// TIA Portal project "Robot_Presantation_Project_V1.0" (V16)

(* hardware
DEVICE "S7-1200 station_1"  S7-1200 Station
   slot 0: "Rack_0"  S7-1200 Rack  Rack  V1.0
   slot 1: "PLC_1"  CPU 1214C DC/DC/DC  6ES7 214-1AG40-0XB0  V4.4
   slot 2: "DI 16/DQ 16x24VDC_1"  6ES7 223-1BL32-0XB0  V2.0
DEVICE "GSD device_1"  GSD.Device.PN
   slot 0: "Rack"  Rack  V1.0
   slot 0: "RC700-PROFINET-IO"  RT RC700_PNIO_V2  RC700-PROFINET-IO  V1.0
      slot 0: "RT RC700_PNIO_V2"  RT RC700_PNIO_V2
      slot 1: "Interface"  Interface
         slot 1: "RJ45 100 MBit/s"  RJ45 100 MBit/s
   slot 1: "Output 32 bytes_1"  Output 32 bytes
      slot 0: "Output 32 bytes"  Output 32 bytes
   slot 2: "Input 32 bytes_1"  Input 32 bytes
      slot 0: "Input 32 bytes"  Input 32 bytes
*)

// ===== PLC "PLC_1"  CPU 1214C DC/DC/DC =====

VAR_GLOBAL   // PLC tag table "Default tag table"
   "Processing Request" AT %M0.0 : Bool;
   "Button_Led_1" AT %Q0.0 : Bool;
   "Permission_To_Send_Response" AT %M0.1 : Bool;
   "Video_Done_Playing" AT %M50.0 : Bool;
   "Tag_3" AT %M1.0 : Bool;
   "Tag_4" AT %M100.0 : Bool;
   "ROBOT_1_READY" AT %M200.0 : Bool;
   "PLC_Enable_Procedures" AT %M2.0 : Bool;
   "Permission_To_Write_To_PC" AT %M3.0 : Bool;
   "Error_On_Communication" AT %M5.0 : Bool;
   "Reset_Error_On_Communication" AT %M5.1 : Bool;
   "Button_1" AT %I0.0 : Bool;
   "Tag_1" AT %M50.1 : Bool;
   "Button_2" AT %I0.1 : Bool;
   "Button_Led_2" AT %Q0.1 : Bool;
   "Button_3" AT %I0.2 : Bool;
   "Button_Led_3" AT %Q0.2 : Bool;
   "TEST_BIT_ROBOT_1_AT_POSITION" AT %M500.0 : Bool;
   "TEST_BIT_ROBOT_1_AT_HOME" AT %M500.1 : Bool;
   "Virtual Button 1" AT %M600.0 : Bool;
   "Tag_7" AT %M6000.0 : Bool;
   "Toggle_test_Bit_Robot_1_At_position" AT %M500.2 : Bool;
   "ROBOT_AT_POSITION_ID_TEMP" AT %MW33 : Int;
   "Robot_2_Ready" AT %M200.1 : Bool;
   "Enable_Robots" AT %M700.0 : Bool;
   "ROBOT_2_AT_POSITION_ID_TEMP" AT %MW35 : Int;
   "System_Byte" AT %MB299 : Byte;
   "FirstScan" AT %M299.0 : Bool;
   "DiagStatusUpdate" AT %M299.1 : Bool;
   "AlwaysTRUE" AT %M299.2 : Bool;
   "AlwaysFALSE" AT %M299.3 : Bool;
   "Clock_Byte" AT %MB298 : Byte;
   "Clock_10Hz" AT %M298.0 : Bool;
   "Clock_5Hz" AT %M298.1 : Bool;
   "Clock_2.5Hz" AT %M298.2 : Bool;
   "Clock_2Hz" AT %M298.3 : Bool;
   "Clock_1.25Hz" AT %M298.4 : Bool;
   "Clock_1Hz" AT %M298.5 : Bool;
   "Clock_0.625Hz" AT %M298.6 : Bool;
   "Clock_0.5Hz" AT %M298.7 : Bool;
   "Button_4" AT %I0.3 : Bool;
   "Button_5" AT %I0.4 : Bool;
   "Button_6" AT %I0.5 : Bool;
   "Button_7" AT %I0.6 : Bool;
   "Button_8" AT %I0.7 : Bool;
   "Button_9" AT %I1.0 : Bool;
   "Button_10" AT %I1.1 : Bool;
   "Button_11" AT %I1.2 : Bool;
   "Button_12" AT %I1.3 : Bool;
   "Button_13" AT %I1.4 : Bool;
   "Button_14" AT %I1.5 : Bool;
   "Button_15" AT %I1.6 : Bool;
   "Button_16" AT %I1.7 : Bool;
   "Button_17" AT %I2.0 : Bool;
   "Button_18" AT %I2.1 : Bool;
   "Button_Led_4" AT %Q0.3 : Bool;
   "Button_Led_5" AT %Q0.4 : Bool;
   "Button_Led_6" AT %Q0.5 : Bool;
   "Button_Led_7" AT %Q0.6 : Bool;
   "Button_Led_8" AT %Q0.7 : Bool;
   "Button_Led_9" AT %Q1.0 : Bool;
   "Button_Led_10" AT %Q1.1 : Bool;
   "Button_Led_11" AT %Q1.2 : Bool;
   "Button_Led_12" AT %Q1.3 : Bool;
   "Button_Led_13" AT %Q1.4 : Bool;
   "Button_Led_14" AT %Q1.5 : Bool;
   "Button_Led_15" AT %Q1.6 : Bool;
   "Button_Led_16" AT %Q1.7 : Bool;
   "Button_Led_17" AT %Q2.0 : Bool;
   "Button_Led_18" AT %Q2.1 : Bool;
   "Robot_Doors_Latched" AT %M700.1 : Bool;
   "Robot_Latch_Doors" AT %Q3.7 : Bool;
   "Input_Data1_From_Robot" AT %IW68 : Word;
   "Input_Data2_From_Robot" AT %IW70 : Word;
   "Input_Data3_From_Robot" AT %IW72 : Word;
   "Input_Data4_From_Robot" AT %IW74 : Word;
   "Output_Data1_To_Robot" AT %QW64 : Word;
   "Output_Data2_To_Robot" AT %QW66 : Word;
   "Output_Data3_To_Robot" AT %QW68 : Word;
   "EMG_OK" AT %I3.7 : Bool;
   "Robot_Reset_Done" AT %M700.2 : Bool;
   "Robot_HOME_OK" AT %M700.3 : Bool;
   "Tag_2" AT %M1003.0 : Bool;
   "Tag_5" AT %M8000.0 : Bool;
   "Virtual Button 2" AT %M600.1 : Bool;
   "Virtual Button 3" AT %M600.2 : Bool;
   "Virtual Button  4" AT %M600.3 : Bool;
   "Virtual Button 5" AT %M600.4 : Bool;
   "Virtual Button 6" AT %M600.5 : Bool;
   "Virtual Button 7" AT %M6000.6 : Bool;
   "Virtual Button 8" AT %M600.7 : Bool;
   "Virtual Button 9" AT %M601.0 : Bool;
   "Virtual Button 10" AT %M601.1 : Bool;
   "Virtual Button 11" AT %M601.2 : Bool;
   "Virtual Button 12" AT %M601.3 : Bool;
   "Virtual Button 13" AT %M601.4 : Bool;
   "Virtual Button 14" AT %M601.5 : Bool;
   "Virtual Button 15" AT %M601.6 : Bool;
   "Virtual Button 16" AT %M601.7 : Bool;
   "Virtual Button 17" AT %M602.0 : Bool;
   "Virtual Button 18" AT %M602.1 : Bool;
   "Enable All Virtual Buttons" AT %M602.2 : Bool;
END_VAR

DATA_BLOCK "PLC_PC_Handshake"   // DB1
{ S7_Optimized_Access := 'FALSE' }
VERSION : 0.1
   VAR
      PC_To_PLC_Request_Connection : Bool;
      PLC_To_PC_Response_Connection : Bool;
      PC_Ready : Bool;
      PC_Busy : Bool;
      PLC_To_PC_Ready_To_Play_Video_Robot_1 : Bool;
      TestConnection : Bool;
      Connection_To_PC_Lost : Bool;
      PC_To_PLC_Video_Playing_Robot_1 : Bool;
      PC_To_PLC_Video_Done_Playing_Robot_1 : Bool;
      PC_To_PLC_Video_Playing_Robot_2 : Bool;
      PC_To_PLC_Video_Done_Playing_Robot_2 : Bool;
      Buffer_Array_Robot_1 : Array[0..19] of Int;
      Buffer_Array_Robot_2 : Array[0..19] of Int;
      PLC_To_PC_Ready_To_Play_Video_Robot_2 : Bool;
      Empty_Array : Array[0..19] of Int;
   END_VAR
BEGIN
END_DATA_BLOCK

DATA_BLOCK "DB_Robot"   // DB45
{ S7_Optimized_Access := 'FALSE' }
VERSION : 0.1
   VAR
      Ready : Bool;
      Running : Bool;
      Paused : Bool;
      Error : Bool;
      Warning : Bool;
      Inside_Box1 : Bool;
      Inside_Box2 : Bool;
      Inside_Box3 : Bool;
      s1 : Bool;
      s2 : Bool;
      s3 : Bool;
      s4 : Bool;
      s5 : Bool;
      s6 : Bool;
      s7 : Bool;
      s8 : Bool;
      At_Position_ID_Robot_1 : Word;
      ErrorID : Word;
      At_Position_ID_Robot_2 : Word;
      Start : Bool;
      Pause : Bool;
      Continue : Bool;
      Reset : Bool;
      Spare_Out1 : Bool;
      Spare_Out2 : Bool;
      Spare_Out3 : Bool;
      Spare_Out4 : Bool;
      Spare_Out5 : Bool;
      Spare_Out6 : Bool;
      Spare_Out7 : Bool;
      Spare_Out8 : Bool;
      Spare_Out9 : Bool;
      Spare_Out10 : Bool;
      Spare_Out11 : Bool;
      Spare_Out12 : Bool;
      To_Position_ID_Robot_1 : Word;
      To_Position_ID_Robot_2 : Word;
   END_VAR
BEGIN
END_DATA_BLOCK

// folder: DBs From FB

DATA_BLOCK "Button_Number_1"   // DB5
{ S7_Optimized_Access := 'TRUE' }
VERSION : 0.1
// stored: InstanceOfName onButton_Press
"onButton_Press"
BEGIN
END_DATA_BLOCK

DATA_BLOCK "Button_Number_2"   // DB8
{ S7_Optimized_Access := 'TRUE' }
VERSION : 0.1
// stored: InstanceOfName onButton_Press
"onButton_Press"
BEGIN
END_DATA_BLOCK

DATA_BLOCK "Button_Number_3"   // DB10
{ S7_Optimized_Access := 'TRUE' }
VERSION : 0.1
// stored: InstanceOfName onButton_Press
"onButton_Press"
BEGIN
END_DATA_BLOCK

DATA_BLOCK "Robot_1_Control"   // DB11
{ S7_Optimized_Access := 'TRUE' }
VERSION : 0.1
// stored: InstanceOfName Robot_Control
"Robot_Control"
BEGIN
END_DATA_BLOCK

DATA_BLOCK "Robot_2_Control"   // DB12
{ S7_Optimized_Access := 'TRUE' }
VERSION : 0.1
// stored: InstanceOfName Robot_Control
"Robot_Control"
BEGIN
END_DATA_BLOCK

DATA_BLOCK "Button_Number_4"   // DB20
{ S7_Optimized_Access := 'TRUE' }
VERSION : 0.1
// stored: InstanceOfName onButton_Press
"onButton_Press"
BEGIN
END_DATA_BLOCK

DATA_BLOCK "Button_Number_5"   // DB21
{ S7_Optimized_Access := 'TRUE' }
VERSION : 0.1
// stored: InstanceOfName onButton_Press
"onButton_Press"
BEGIN
END_DATA_BLOCK

DATA_BLOCK "Button_Number_6"   // DB22
{ S7_Optimized_Access := 'TRUE' }
VERSION : 0.1
// stored: InstanceOfName onButton_Press
"onButton_Press"
BEGIN
END_DATA_BLOCK

DATA_BLOCK "Button_Number_7"   // DB23
{ S7_Optimized_Access := 'TRUE' }
VERSION : 0.1
// stored: InstanceOfName onButton_Press
"onButton_Press"
BEGIN
END_DATA_BLOCK

DATA_BLOCK "Button_Number_8"   // DB24
{ S7_Optimized_Access := 'TRUE' }
VERSION : 0.1
// stored: InstanceOfName onButton_Press
"onButton_Press"
BEGIN
END_DATA_BLOCK

DATA_BLOCK "Button_Number_9"   // DB25
{ S7_Optimized_Access := 'TRUE' }
VERSION : 0.1
// stored: InstanceOfName onButton_Press
"onButton_Press"
BEGIN
END_DATA_BLOCK

DATA_BLOCK "Button_Number_10"   // DB26
{ S7_Optimized_Access := 'TRUE' }
VERSION : 0.1
// stored: InstanceOfName onButton_Press
"onButton_Press"
BEGIN
END_DATA_BLOCK

DATA_BLOCK "Button_Number_11"   // DB28
{ S7_Optimized_Access := 'TRUE' }
VERSION : 0.1
// stored: InstanceOfName onButton_Press
"onButton_Press"
BEGIN
END_DATA_BLOCK

DATA_BLOCK "Button_Number_12"   // DB30
{ S7_Optimized_Access := 'TRUE' }
VERSION : 0.1
// stored: InstanceOfName onButton_Press
"onButton_Press"
BEGIN
END_DATA_BLOCK

DATA_BLOCK "Button_Number_13"   // DB32
{ S7_Optimized_Access := 'TRUE' }
VERSION : 0.1
// stored: InstanceOfName onButton_Press
"onButton_Press"
BEGIN
END_DATA_BLOCK

DATA_BLOCK "Button_Number_14"   // DB34
{ S7_Optimized_Access := 'TRUE' }
VERSION : 0.1
// stored: InstanceOfName onButton_Press
"onButton_Press"
BEGIN
END_DATA_BLOCK

DATA_BLOCK "Button_Number_15"   // DB36
{ S7_Optimized_Access := 'TRUE' }
VERSION : 0.1
// stored: InstanceOfName onButton_Press
"onButton_Press"
BEGIN
END_DATA_BLOCK

DATA_BLOCK "Button_Number_16"   // DB38
{ S7_Optimized_Access := 'TRUE' }
VERSION : 0.1
// stored: InstanceOfName onButton_Press
"onButton_Press"
BEGIN
END_DATA_BLOCK

DATA_BLOCK "Button_Number_17"   // DB40
{ S7_Optimized_Access := 'TRUE' }
VERSION : 0.1
// stored: InstanceOfName onButton_Press
"onButton_Press"
BEGIN
END_DATA_BLOCK

DATA_BLOCK "Button_Number_18"   // DB42
{ S7_Optimized_Access := 'TRUE' }
VERSION : 0.1
// stored: InstanceOfName onButton_Press
"onButton_Press"
BEGIN
END_DATA_BLOCK

// folder: System blocks/Program resources

DATA_BLOCK "TON_TestConnection_On_Signal"   // DB3
{ S7_Optimized_Access := 'TRUE' }
AUTHOR : Simatic
FAMILY : IEC
NAME : IEC_TMR
VERSION : 1.0
// stored: InstanceOfName IEC_TIMER
"IEC_TIMER"
BEGIN
END_DATA_BLOCK

DATA_BLOCK "TON_TestConnection_Off_Signal"   // DB4
{ S7_Optimized_Access := 'TRUE' }
AUTHOR : Simatic
FAMILY : IEC
NAME : IEC_TMR
VERSION : 1.0
// stored: InstanceOfName IEC_TIMER
"IEC_TIMER"
BEGIN
END_DATA_BLOCK

DATA_BLOCK "Test_Timer_Sequence_1"   // DB6
{ S7_Optimized_Access := 'TRUE' }
AUTHOR : Simatic
FAMILY : IEC
NAME : IEC_TMR
VERSION : 1.0
// stored: InstanceOfName IEC_TIMER
"IEC_TIMER"
BEGIN
END_DATA_BLOCK

DATA_BLOCK "Test_Timer_Sequence_2"   // DB7
{ S7_Optimized_Access := 'TRUE' }
AUTHOR : Simatic
FAMILY : IEC
NAME : IEC_TMR
VERSION : 1.0
// stored: InstanceOfName IEC_TIMER
"IEC_TIMER"
BEGIN
END_DATA_BLOCK

DATA_BLOCK "Test_Timer_Sequence_3"   // DB9
{ S7_Optimized_Access := 'TRUE' }
AUTHOR : Simatic
FAMILY : IEC
NAME : IEC_TMR
VERSION : 1.0
// stored: InstanceOfName IEC_TIMER
"IEC_TIMER"
BEGIN
END_DATA_BLOCK

DATA_BLOCK "Enable_PLC_PC_Comms"   // DB13
{ S7_Optimized_Access := 'TRUE' }
AUTHOR : Simatic
FAMILY : IEC
NAME : IEC_TMR
VERSION : 1.0
// stored: InstanceOfName IEC_TIMER
"IEC_TIMER"
BEGIN
END_DATA_BLOCK

DATA_BLOCK "Test_Timer_Sequence_4"   // DB14
{ S7_Optimized_Access := 'TRUE' }
AUTHOR : Simatic
FAMILY : IEC
NAME : IEC_TMR
VERSION : 1.0
// stored: InstanceOfName IEC_TIMER
"IEC_TIMER"
BEGIN
END_DATA_BLOCK

DATA_BLOCK "Test_Timer_Sequence_5"   // DB15
{ S7_Optimized_Access := 'TRUE' }
AUTHOR : Simatic
FAMILY : IEC
NAME : IEC_TMR
VERSION : 1.0
// stored: InstanceOfName IEC_TIMER
"IEC_TIMER"
BEGIN
END_DATA_BLOCK

DATA_BLOCK "Test_Timer_Sequence_6"   // DB16
{ S7_Optimized_Access := 'TRUE' }
AUTHOR : Simatic
FAMILY : IEC
NAME : IEC_TMR
VERSION : 1.0
// stored: InstanceOfName IEC_TIMER
"IEC_TIMER"
BEGIN
END_DATA_BLOCK

DATA_BLOCK "Test_Timer_Sequence_7"   // DB17
{ S7_Optimized_Access := 'TRUE' }
AUTHOR : Simatic
FAMILY : IEC
NAME : IEC_TMR
VERSION : 1.0
// stored: InstanceOfName IEC_TIMER
"IEC_TIMER"
BEGIN
END_DATA_BLOCK

DATA_BLOCK "Test_Timer_Sequence_8"   // DB18
{ S7_Optimized_Access := 'TRUE' }
AUTHOR : Simatic
FAMILY : IEC
NAME : IEC_TMR
VERSION : 1.0
// stored: InstanceOfName IEC_TIMER
"IEC_TIMER"
BEGIN
END_DATA_BLOCK

DATA_BLOCK "Test_Timer_Sequence_9"   // DB19
{ S7_Optimized_Access := 'TRUE' }
AUTHOR : Simatic
FAMILY : IEC
NAME : IEC_TMR
VERSION : 1.0
// stored: InstanceOfName IEC_TIMER
"IEC_TIMER"
BEGIN
END_DATA_BLOCK

DATA_BLOCK "Test_Timer_Sequence_10"   // DB27
{ S7_Optimized_Access := 'TRUE' }
AUTHOR : Simatic
FAMILY : IEC
NAME : IEC_TMR
VERSION : 1.0
// stored: InstanceOfName IEC_TIMER
"IEC_TIMER"
BEGIN
END_DATA_BLOCK

DATA_BLOCK "Test_Timer_Sequence_11"   // DB29
{ S7_Optimized_Access := 'TRUE' }
AUTHOR : Simatic
FAMILY : IEC
NAME : IEC_TMR
VERSION : 1.0
// stored: InstanceOfName IEC_TIMER
"IEC_TIMER"
BEGIN
END_DATA_BLOCK

DATA_BLOCK "Test_Timer_Sequence_12"   // DB31
{ S7_Optimized_Access := 'TRUE' }
AUTHOR : Simatic
FAMILY : IEC
NAME : IEC_TMR
VERSION : 1.0
// stored: InstanceOfName IEC_TIMER
"IEC_TIMER"
BEGIN
END_DATA_BLOCK

DATA_BLOCK "Test_Timer_Sequence_13"   // DB33
{ S7_Optimized_Access := 'TRUE' }
AUTHOR : Simatic
FAMILY : IEC
NAME : IEC_TMR
VERSION : 1.0
// stored: InstanceOfName IEC_TIMER
"IEC_TIMER"
BEGIN
END_DATA_BLOCK

DATA_BLOCK "Test_Timer_Sequence_14"   // DB35
{ S7_Optimized_Access := 'TRUE' }
AUTHOR : Simatic
FAMILY : IEC
NAME : IEC_TMR
VERSION : 1.0
// stored: InstanceOfName IEC_TIMER
"IEC_TIMER"
BEGIN
END_DATA_BLOCK

DATA_BLOCK "Test_Timer_Sequence_15"   // DB37
{ S7_Optimized_Access := 'TRUE' }
AUTHOR : Simatic
FAMILY : IEC
NAME : IEC_TMR
VERSION : 1.0
// stored: InstanceOfName IEC_TIMER
"IEC_TIMER"
BEGIN
END_DATA_BLOCK

DATA_BLOCK "Test_Timer_Sequence_16"   // DB39
{ S7_Optimized_Access := 'TRUE' }
AUTHOR : Simatic
FAMILY : IEC
NAME : IEC_TMR
VERSION : 1.0
// stored: InstanceOfName IEC_TIMER
"IEC_TIMER"
BEGIN
END_DATA_BLOCK

DATA_BLOCK "Test_Timer_Sequence_17"   // DB41
{ S7_Optimized_Access := 'TRUE' }
AUTHOR : Simatic
FAMILY : IEC
NAME : IEC_TMR
VERSION : 1.0
// stored: InstanceOfName IEC_TIMER
"IEC_TIMER"
BEGIN
END_DATA_BLOCK

DATA_BLOCK "Test_Timer_Sequence_18"   // DB43
{ S7_Optimized_Access := 'TRUE' }
AUTHOR : Simatic
FAMILY : IEC
NAME : IEC_TMR
VERSION : 1.0
// stored: InstanceOfName IEC_TIMER
"IEC_TIMER"
BEGIN
END_DATA_BLOCK

DATA_BLOCK "TON_Robot_Latch_Doors"   // DB44
{ S7_Optimized_Access := 'TRUE' }
AUTHOR : Simatic
FAMILY : IEC
NAME : IEC_TMR
VERSION : 1.0
// stored: InstanceOfName IEC_TIMER
"IEC_TIMER"
BEGIN
END_DATA_BLOCK

DATA_BLOCK "TON_Timer_Robot_To_Reset"   // DB46
{ S7_Optimized_Access := 'TRUE' }
AUTHOR : Simatic
FAMILY : IEC
NAME : IEC_TMR
VERSION : 1.0
// stored: InstanceOfName IEC_TIMER
"IEC_TIMER"
BEGIN
END_DATA_BLOCK

DATA_BLOCK "TON_Timer_Robot_Reset"   // DB47
{ S7_Optimized_Access := 'TRUE' }
AUTHOR : Simatic
FAMILY : IEC
NAME : IEC_TMR
VERSION : 1.0
// stored: InstanceOfName IEC_TIMER
"IEC_TIMER"
BEGIN
END_DATA_BLOCK

DATA_BLOCK "TON_Timer_To_Start_Robot"   // DB48
{ S7_Optimized_Access := 'TRUE' }
AUTHOR : Simatic
FAMILY : IEC
NAME : IEC_TMR
VERSION : 1.0
// stored: InstanceOfName IEC_TIMER
"IEC_TIMER"
BEGIN
END_DATA_BLOCK

DATA_BLOCK "TON_Robot_Start_Delay"   // DB49
{ S7_Optimized_Access := 'TRUE' }
AUTHOR : Simatic
FAMILY : IEC
NAME : IEC_TMR
VERSION : 1.0
// stored: InstanceOfName IEC_TIMER
"IEC_TIMER"
BEGIN
END_DATA_BLOCK

// folder: (top level)

FUNCTION "PC_PLC_Connection" : Void   // FC1, LAD
{ S7_Optimized_Access := 'TRUE' }
VERSION : 0.1
BEGIN

REGION Network 1: PC requesting to connect, PLC response with bit
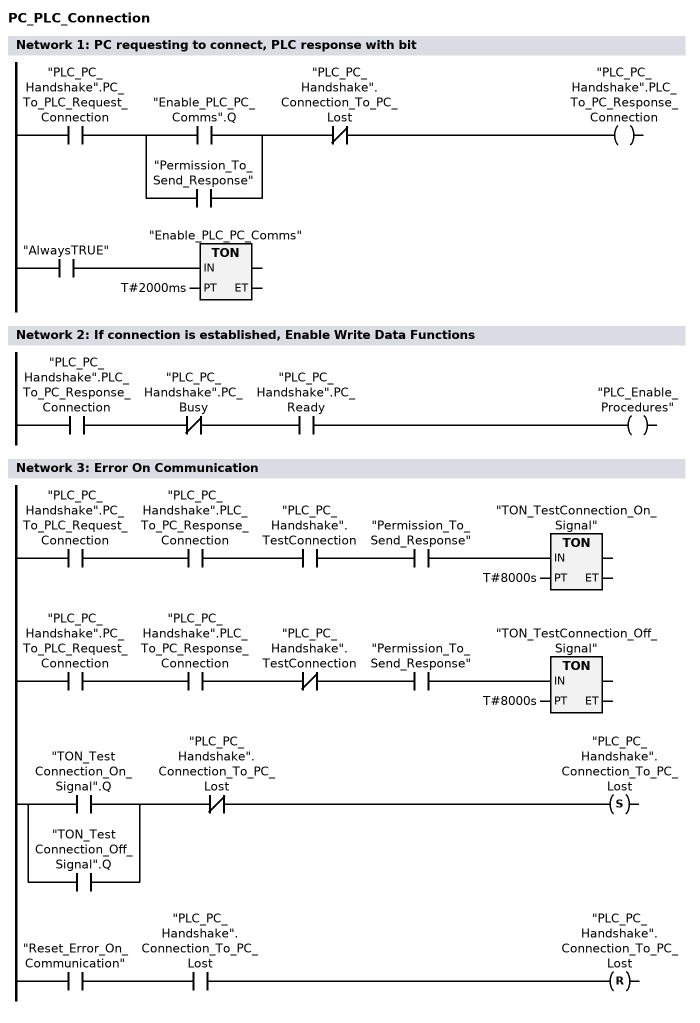
   "PLC_PC_Handshake".PLC_To_PC_Response_Connection := "PLC_PC_Handshake".PC_To_PLC_Request_Connection AND ("Enable_PLC_PC_Comms".Q OR "Permission_To_Send_Response") AND NOT "PLC_PC_Handshake".Connection_To_PC_Lost;
   "Enable_PLC_PC_Comms".TON(IN := "AlwaysTRUE", PT := T#2000ms);
END_REGION

REGION Network 2: If connection is established, Enable Write Data Functions
   RUNG wire#powerrail
      Contact( "PLC_PC_Handshake".PLC_To_PC_Response_Connection )
      I_Contact( "PLC_PC_Handshake".PC_Busy )
      Contact( "PLC_PC_Handshake".PC_Ready )
      Coil( "PLC_Enable_Procedures" )
   END_RUNG
   // the same network as SCL:
   "PLC_Enable_Procedures" := "PLC_PC_Handshake".PLC_To_PC_Response_Connection AND NOT "PLC_PC_Handshake".PC_Busy AND "PLC_PC_Handshake".PC_Ready;
END_REGION

REGION Network 3: Error On Communication
   "TON_TestConnection_On_Signal".TON(IN := "PLC_PC_Handshake".PC_To_PLC_Request_Connection AND "PLC_PC_Handshake".PLC_To_PC_Response_Connection AND "PLC_PC_Handshake".TestConnection AND "Permission_To_Send_Response",
                           PT := T#8000s);
   "TON_TestConnection_Off_Signal".TON(IN := "PLC_PC_Handshake".PC_To_PLC_Request_Connection AND "PLC_PC_Handshake".PLC_To_PC_Response_Connection AND NOT "PLC_PC_Handshake".TestConnection AND "Permission_To_Send_Response",
                           PT := T#8000s);
   IF ("TON_TestConnection_On_Signal".Q OR "TON_TestConnection_Off_Signal".Q) AND NOT "PLC_PC_Handshake".Connection_To_PC_Lost THEN
       "PLC_PC_Handshake".Connection_To_PC_Lost := TRUE;
   END_IF;
   IF "Reset_Error_On_Communication" AND "PLC_PC_Handshake".Connection_To_PC_Lost THEN
       "PLC_PC_Handshake".Connection_To_PC_Lost := FALSE;
   END_IF;
END_REGION
END_FUNCTION

FUNCTION "Buttons_Functionality" : Void   // FC2, LAD
{ S7_Optimized_Access := 'TRUE' }
VERSION : 0.1
BEGIN

REGION Network 1: Button 1, Robot 1, Position ID 10
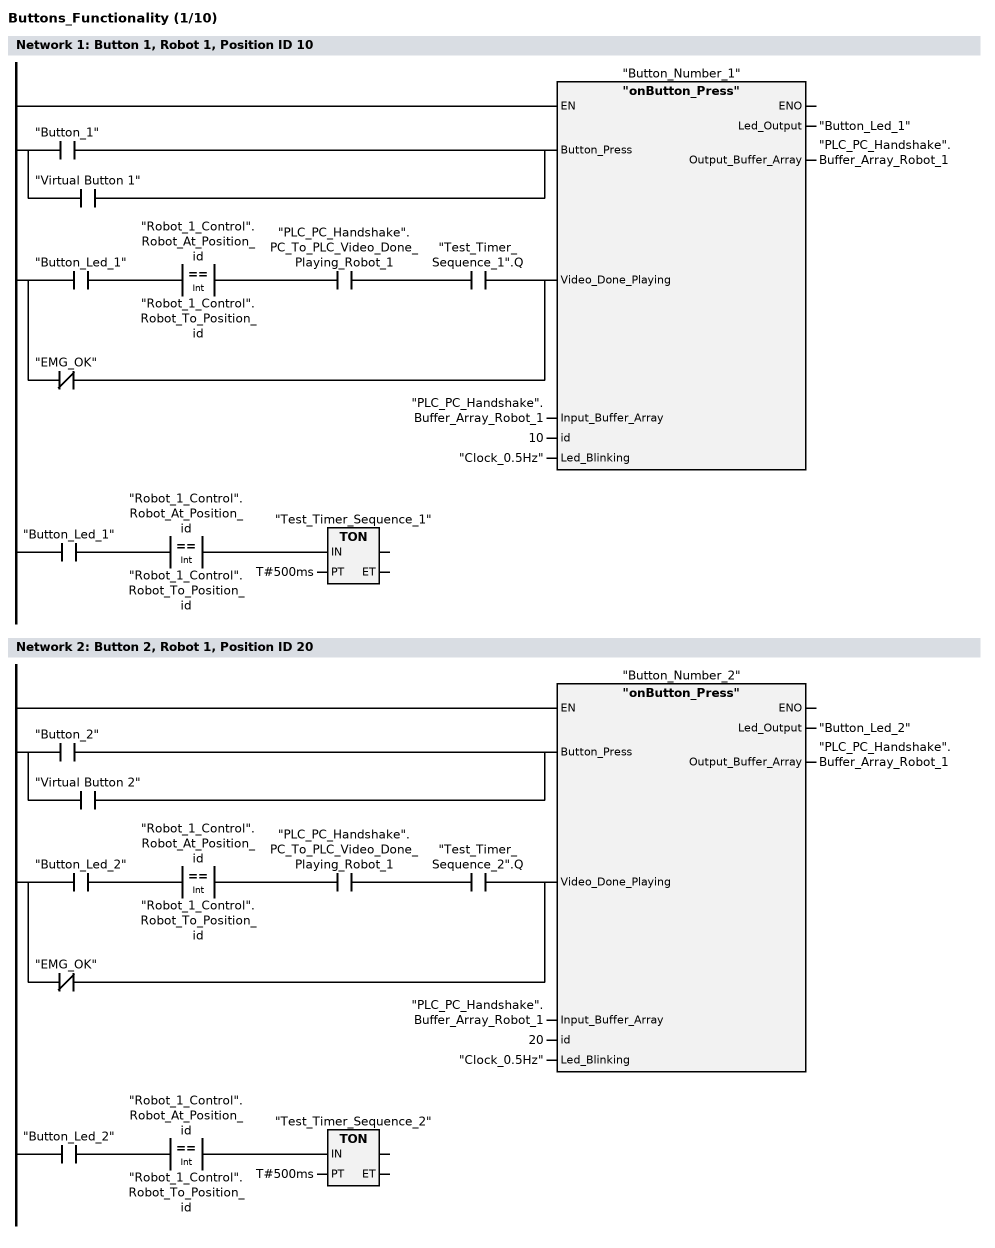
   "Button_Number_1"(Button_Press := "Button_1" OR "Virtual Button 1",   // "onButton_Press"
                     Video_Done_Playing := ("Button_Led_1" AND ("Robot_1_Control".Robot_At_Position_id = "Robot_1_Control".Robot_To_Position_id) AND "PLC_PC_Handshake".PC_To_PLC_Video_Done_Playing_Robot_1 AND "Test_Timer_Sequence_1".Q) OR NOT "EMG_OK",
                     Input_Buffer_Array := "PLC_PC_Handshake".Buffer_Array_Robot_1,
                     id := 10,
                     Led_Blinking := "Clock_0.5Hz",
                     Led_Output => "Button_Led_1",
                     Output_Buffer_Array => "PLC_PC_Handshake".Buffer_Array_Robot_1);
   "Test_Timer_Sequence_1".TON(IN := "Button_Led_1" AND ("Robot_1_Control".Robot_At_Position_id = "Robot_1_Control".Robot_To_Position_id),
                           PT := T#500ms);
END_REGION

REGION Network 2: Button 2, Robot 1, Position ID 20
   "Button_Number_2"(Button_Press := "Button_2" OR "Virtual Button 2",   // "onButton_Press"
                     Video_Done_Playing := ("Button_Led_2" AND ("Robot_1_Control".Robot_At_Position_id = "Robot_1_Control".Robot_To_Position_id) AND "PLC_PC_Handshake".PC_To_PLC_Video_Done_Playing_Robot_1 AND "Test_Timer_Sequence_2".Q) OR NOT "EMG_OK",
                     Input_Buffer_Array := "PLC_PC_Handshake".Buffer_Array_Robot_1,
                     id := 20,
                     Led_Blinking := "Clock_0.5Hz",
                     Led_Output => "Button_Led_2",
                     Output_Buffer_Array => "PLC_PC_Handshake".Buffer_Array_Robot_1);
   "Test_Timer_Sequence_2".TON(IN := "Button_Led_2" AND ("Robot_1_Control".Robot_At_Position_id = "Robot_1_Control".Robot_To_Position_id),
                           PT := T#500ms);
END_REGION

REGION Network 3: Button 3, Robot 1, Position ID 30
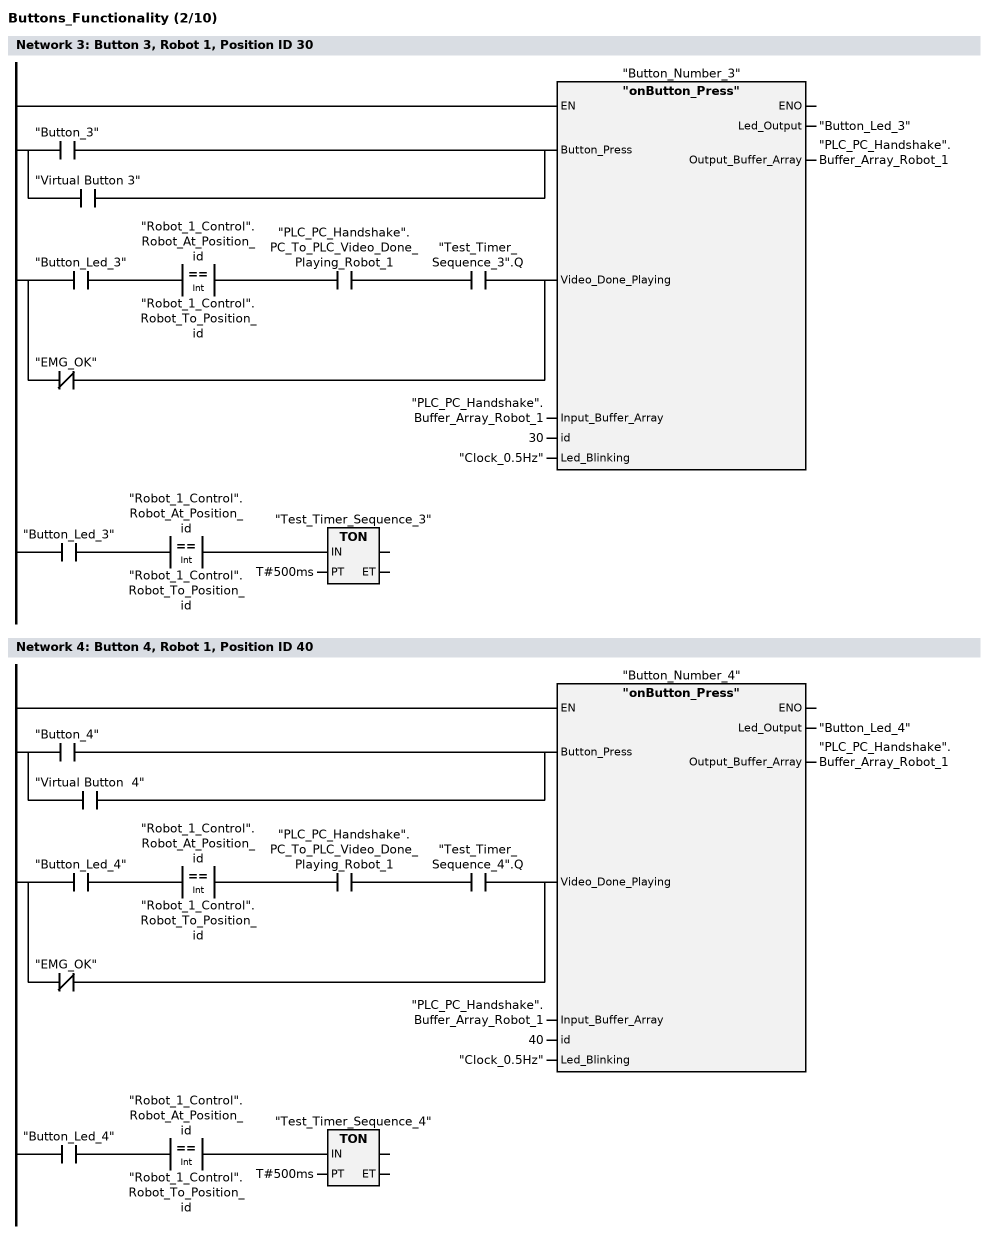
   "Button_Number_3"(Button_Press := "Button_3" OR "Virtual Button 3",   // "onButton_Press"
                     Video_Done_Playing := ("Button_Led_3" AND ("Robot_1_Control".Robot_At_Position_id = "Robot_1_Control".Robot_To_Position_id) AND "PLC_PC_Handshake".PC_To_PLC_Video_Done_Playing_Robot_1 AND "Test_Timer_Sequence_3".Q) OR NOT "EMG_OK",
                     Input_Buffer_Array := "PLC_PC_Handshake".Buffer_Array_Robot_1,
                     id := 30,
                     Led_Blinking := "Clock_0.5Hz",
                     Led_Output => "Button_Led_3",
                     Output_Buffer_Array => "PLC_PC_Handshake".Buffer_Array_Robot_1);
   "Test_Timer_Sequence_3".TON(IN := "Button_Led_3" AND ("Robot_1_Control".Robot_At_Position_id = "Robot_1_Control".Robot_To_Position_id),
                           PT := T#500ms);
END_REGION

REGION Network 4: Button 4, Robot 1, Position ID 40
   "Button_Number_4"(Button_Press := "Button_4" OR "Virtual Button  4",   // "onButton_Press"
                     Video_Done_Playing := ("Button_Led_4" AND ("Robot_1_Control".Robot_At_Position_id = "Robot_1_Control".Robot_To_Position_id) AND "PLC_PC_Handshake".PC_To_PLC_Video_Done_Playing_Robot_1 AND "Test_Timer_Sequence_4".Q) OR NOT "EMG_OK",
                     Input_Buffer_Array := "PLC_PC_Handshake".Buffer_Array_Robot_1,
                     id := 40,
                     Led_Blinking := "Clock_0.5Hz",
                     Led_Output => "Button_Led_4",
                     Output_Buffer_Array => "PLC_PC_Handshake".Buffer_Array_Robot_1);
   "Test_Timer_Sequence_4".TON(IN := "Button_Led_4" AND ("Robot_1_Control".Robot_At_Position_id = "Robot_1_Control".Robot_To_Position_id),
                           PT := T#500ms);
END_REGION

REGION Network 5: Button 5, Robot 1, Position ID 50
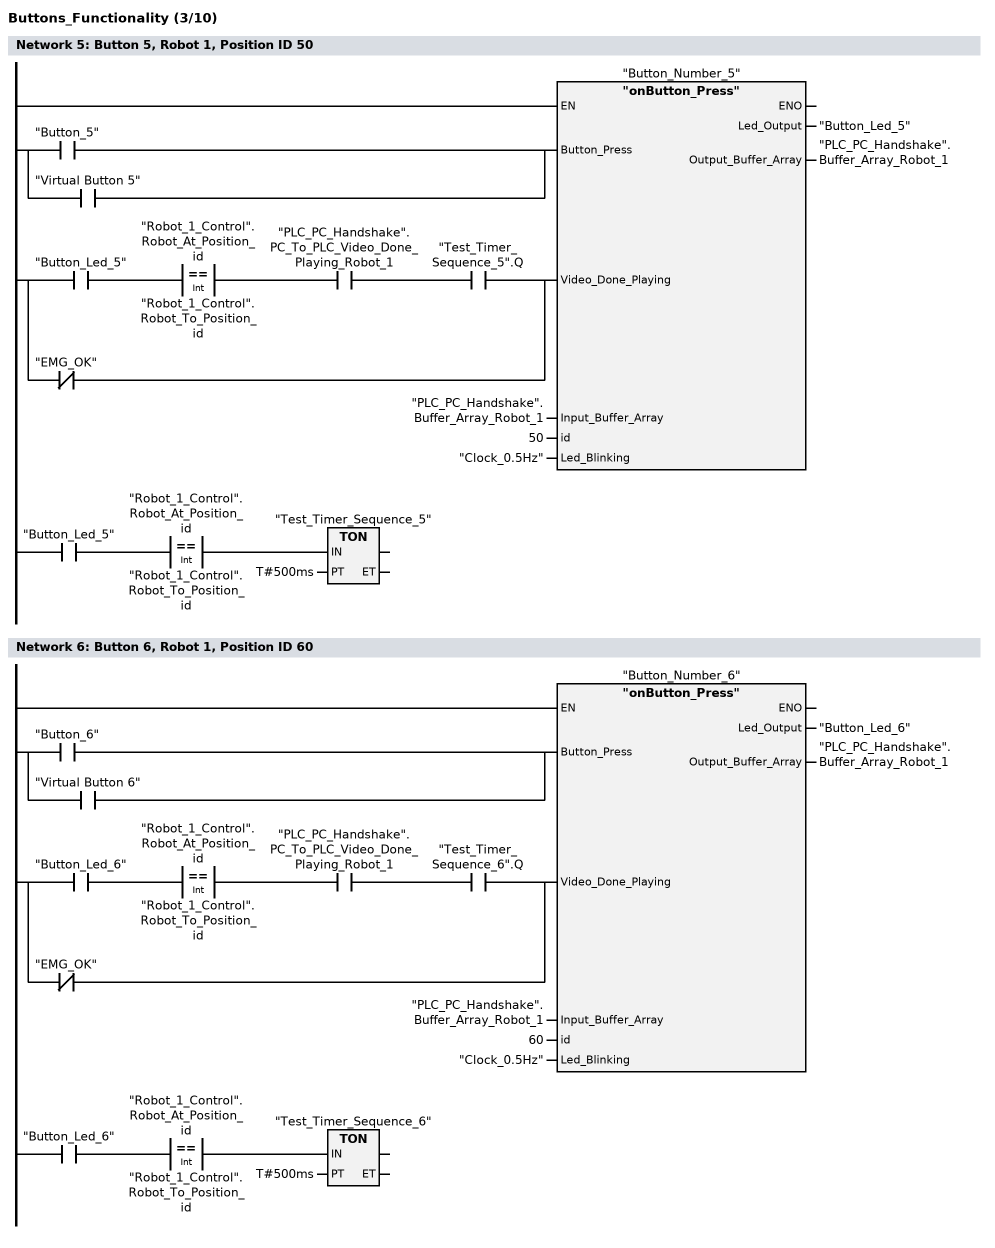
   "Button_Number_5"(Button_Press := "Button_5" OR "Virtual Button 5",   // "onButton_Press"
                     Video_Done_Playing := ("Button_Led_5" AND ("Robot_1_Control".Robot_At_Position_id = "Robot_1_Control".Robot_To_Position_id) AND "PLC_PC_Handshake".PC_To_PLC_Video_Done_Playing_Robot_1 AND "Test_Timer_Sequence_5".Q) OR NOT "EMG_OK",
                     Input_Buffer_Array := "PLC_PC_Handshake".Buffer_Array_Robot_1,
                     id := 50,
                     Led_Blinking := "Clock_0.5Hz",
                     Led_Output => "Button_Led_5",
                     Output_Buffer_Array => "PLC_PC_Handshake".Buffer_Array_Robot_1);
   "Test_Timer_Sequence_5".TON(IN := "Button_Led_5" AND ("Robot_1_Control".Robot_At_Position_id = "Robot_1_Control".Robot_To_Position_id),
                           PT := T#500ms);
END_REGION

REGION Network 6: Button 6, Robot 1, Position ID 60
   "Button_Number_6"(Button_Press := "Button_6" OR "Virtual Button 6",   // "onButton_Press"
                     Video_Done_Playing := ("Button_Led_6" AND ("Robot_1_Control".Robot_At_Position_id = "Robot_1_Control".Robot_To_Position_id) AND "PLC_PC_Handshake".PC_To_PLC_Video_Done_Playing_Robot_1 AND "Test_Timer_Sequence_6".Q) OR NOT "EMG_OK",
                     Input_Buffer_Array := "PLC_PC_Handshake".Buffer_Array_Robot_1,
                     id := 60,
                     Led_Blinking := "Clock_0.5Hz",
                     Led_Output => "Button_Led_6",
                     Output_Buffer_Array => "PLC_PC_Handshake".Buffer_Array_Robot_1);
   "Test_Timer_Sequence_6".TON(IN := "Button_Led_6" AND ("Robot_1_Control".Robot_At_Position_id = "Robot_1_Control".Robot_To_Position_id),
                           PT := T#500ms);
END_REGION

REGION Network 7: Button 7, Robot 1, Position ID 70
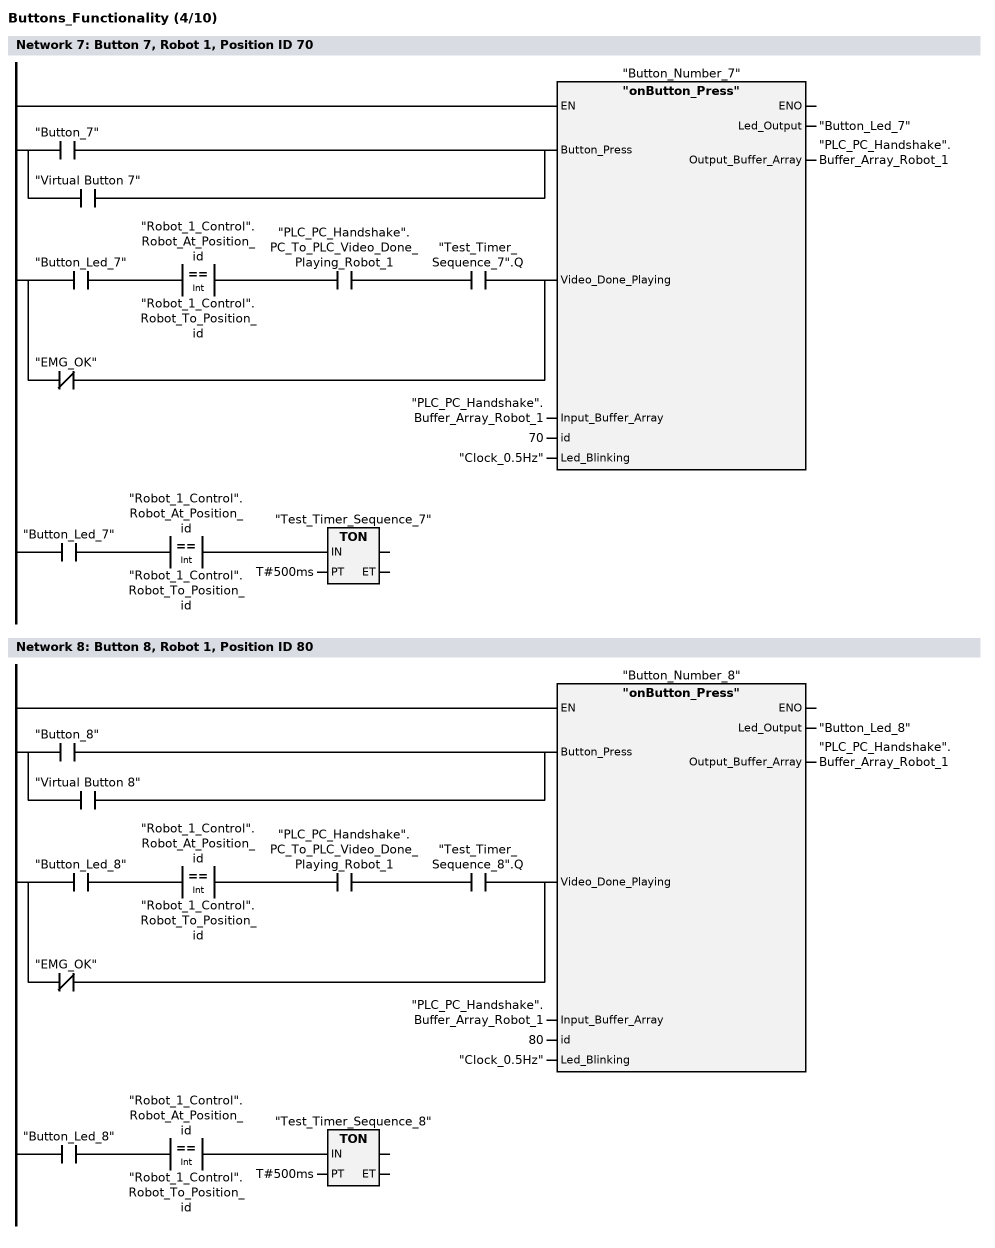
   "Button_Number_7"(Button_Press := "Button_7" OR "Virtual Button 7",   // "onButton_Press"
                     Video_Done_Playing := ("Button_Led_7" AND ("Robot_1_Control".Robot_At_Position_id = "Robot_1_Control".Robot_To_Position_id) AND "PLC_PC_Handshake".PC_To_PLC_Video_Done_Playing_Robot_1 AND "Test_Timer_Sequence_7".Q) OR NOT "EMG_OK",
                     Input_Buffer_Array := "PLC_PC_Handshake".Buffer_Array_Robot_1,
                     id := 70,
                     Led_Blinking := "Clock_0.5Hz",
                     Led_Output => "Button_Led_7",
                     Output_Buffer_Array => "PLC_PC_Handshake".Buffer_Array_Robot_1);
   "Test_Timer_Sequence_7".TON(IN := "Button_Led_7" AND ("Robot_1_Control".Robot_At_Position_id = "Robot_1_Control".Robot_To_Position_id),
                           PT := T#500ms);
END_REGION

REGION Network 8: Button 8, Robot 1, Position ID 80
   "Button_Number_8"(Button_Press := "Button_8" OR "Virtual Button 8",   // "onButton_Press"
                     Video_Done_Playing := ("Button_Led_8" AND ("Robot_1_Control".Robot_At_Position_id = "Robot_1_Control".Robot_To_Position_id) AND "PLC_PC_Handshake".PC_To_PLC_Video_Done_Playing_Robot_1 AND "Test_Timer_Sequence_8".Q) OR NOT "EMG_OK",
                     Input_Buffer_Array := "PLC_PC_Handshake".Buffer_Array_Robot_1,
                     id := 80,
                     Led_Blinking := "Clock_0.5Hz",
                     Led_Output => "Button_Led_8",
                     Output_Buffer_Array => "PLC_PC_Handshake".Buffer_Array_Robot_1);
   "Test_Timer_Sequence_8".TON(IN := "Button_Led_8" AND ("Robot_1_Control".Robot_At_Position_id = "Robot_1_Control".Robot_To_Position_id),
                           PT := T#500ms);
END_REGION

REGION Network 9: Button 9, Robot 1, Position ID 90
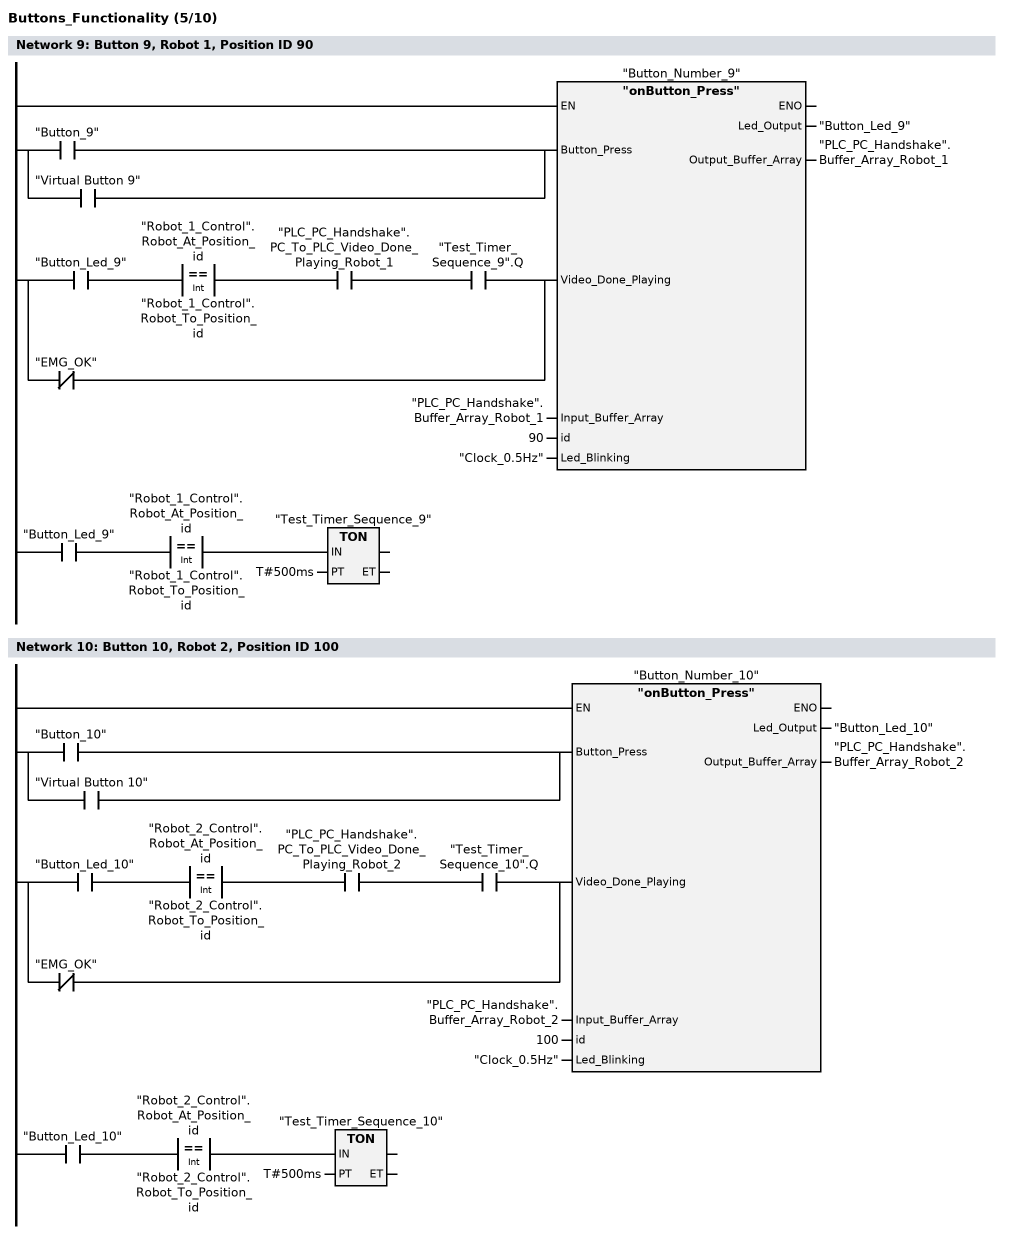
   "Button_Number_9"(Button_Press := "Button_9" OR "Virtual Button 9",   // "onButton_Press"
                     Video_Done_Playing := ("Button_Led_9" AND ("Robot_1_Control".Robot_At_Position_id = "Robot_1_Control".Robot_To_Position_id) AND "PLC_PC_Handshake".PC_To_PLC_Video_Done_Playing_Robot_1 AND "Test_Timer_Sequence_9".Q) OR NOT "EMG_OK",
                     Input_Buffer_Array := "PLC_PC_Handshake".Buffer_Array_Robot_1,
                     id := 90,
                     Led_Blinking := "Clock_0.5Hz",
                     Led_Output => "Button_Led_9",
                     Output_Buffer_Array => "PLC_PC_Handshake".Buffer_Array_Robot_1);
   "Test_Timer_Sequence_9".TON(IN := "Button_Led_9" AND ("Robot_1_Control".Robot_At_Position_id = "Robot_1_Control".Robot_To_Position_id),
                           PT := T#500ms);
END_REGION

REGION Network 10: Button 10, Robot 2, Position ID 100
   "Button_Number_10"(Button_Press := "Button_10" OR "Virtual Button 10",   // "onButton_Press"
                      Video_Done_Playing := ("Button_Led_10" AND ("Robot_2_Control".Robot_At_Position_id = "Robot_2_Control".Robot_To_Position_id) AND "PLC_PC_Handshake".PC_To_PLC_Video_Done_Playing_Robot_2 AND "Test_Timer_Sequence_10".Q) OR NOT "EMG_OK",
                      Input_Buffer_Array := "PLC_PC_Handshake".Buffer_Array_Robot_2,
                      id := 100,
                      Led_Blinking := "Clock_0.5Hz",
                      Led_Output => "Button_Led_10",
                      Output_Buffer_Array => "PLC_PC_Handshake".Buffer_Array_Robot_2);
   "Test_Timer_Sequence_10".TON(IN := "Button_Led_10" AND ("Robot_2_Control".Robot_At_Position_id = "Robot_2_Control".Robot_To_Position_id),
                           PT := T#500ms);
END_REGION

REGION Network 11: Button 11, Robot 2, Position ID 110
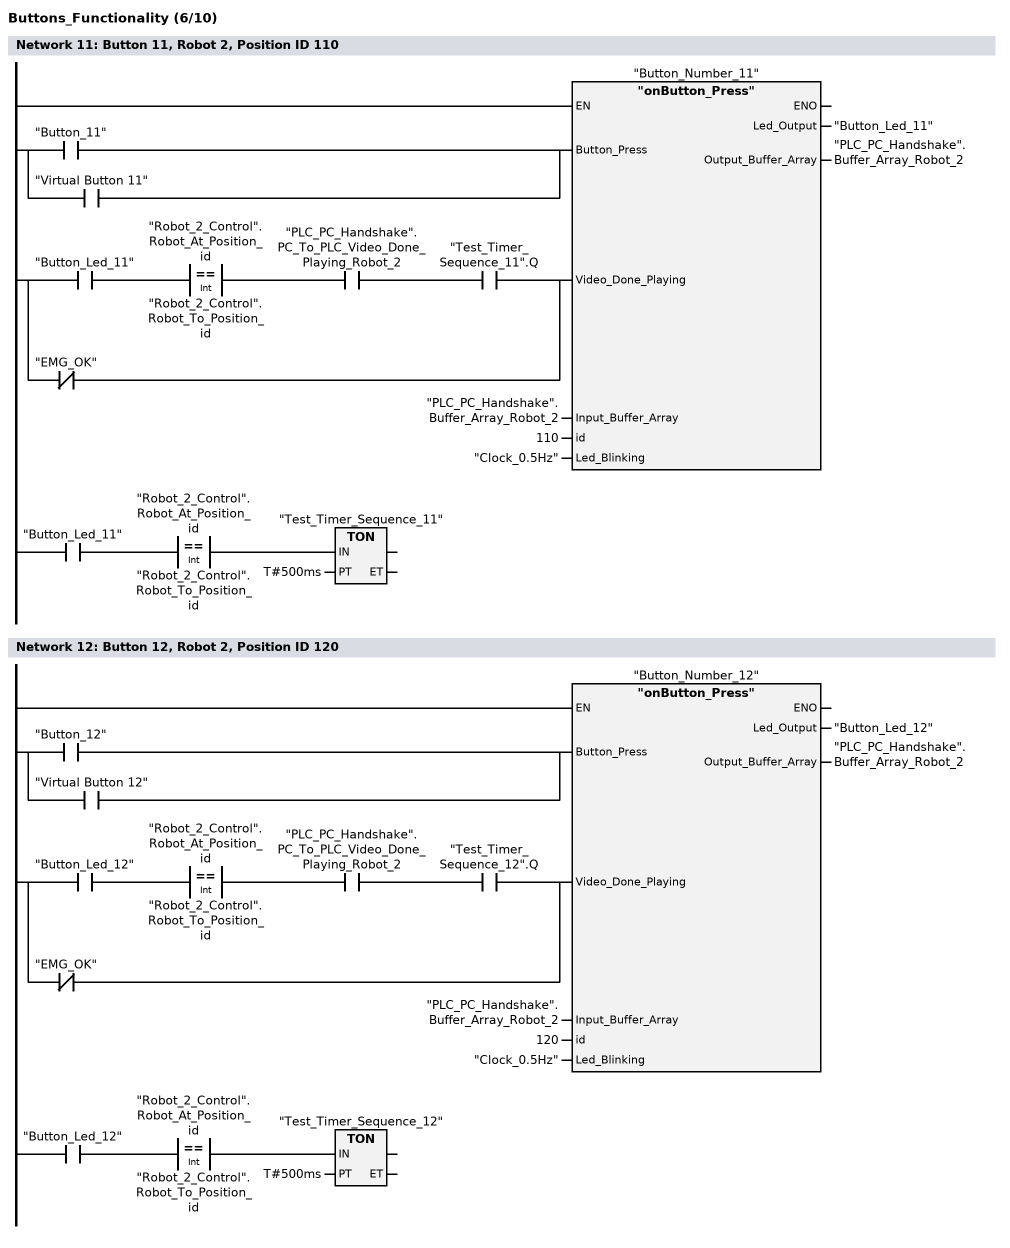
   "Button_Number_11"(Button_Press := "Button_11" OR "Virtual Button 11",   // "onButton_Press"
                      Video_Done_Playing := ("Button_Led_11" AND ("Robot_2_Control".Robot_At_Position_id = "Robot_2_Control".Robot_To_Position_id) AND "PLC_PC_Handshake".PC_To_PLC_Video_Done_Playing_Robot_2 AND "Test_Timer_Sequence_11".Q) OR NOT "EMG_OK",
                      Input_Buffer_Array := "PLC_PC_Handshake".Buffer_Array_Robot_2,
                      id := 110,
                      Led_Blinking := "Clock_0.5Hz",
                      Led_Output => "Button_Led_11",
                      Output_Buffer_Array => "PLC_PC_Handshake".Buffer_Array_Robot_2);
   "Test_Timer_Sequence_11".TON(IN := "Button_Led_11" AND ("Robot_2_Control".Robot_At_Position_id = "Robot_2_Control".Robot_To_Position_id),
                           PT := T#500ms);
END_REGION

REGION Network 12: Button 12, Robot 2, Position ID 120
   "Button_Number_12"(Button_Press := "Button_12" OR "Virtual Button 12",   // "onButton_Press"
                      Video_Done_Playing := ("Button_Led_12" AND ("Robot_2_Control".Robot_At_Position_id = "Robot_2_Control".Robot_To_Position_id) AND "PLC_PC_Handshake".PC_To_PLC_Video_Done_Playing_Robot_2 AND "Test_Timer_Sequence_12".Q) OR NOT "EMG_OK",
                      Input_Buffer_Array := "PLC_PC_Handshake".Buffer_Array_Robot_2,
                      id := 120,
                      Led_Blinking := "Clock_0.5Hz",
                      Led_Output => "Button_Led_12",
                      Output_Buffer_Array => "PLC_PC_Handshake".Buffer_Array_Robot_2);
   "Test_Timer_Sequence_12".TON(IN := "Button_Led_12" AND ("Robot_2_Control".Robot_At_Position_id = "Robot_2_Control".Robot_To_Position_id),
                           PT := T#500ms);
END_REGION

REGION Network 13: Button 13, Robot 2, Position ID 130
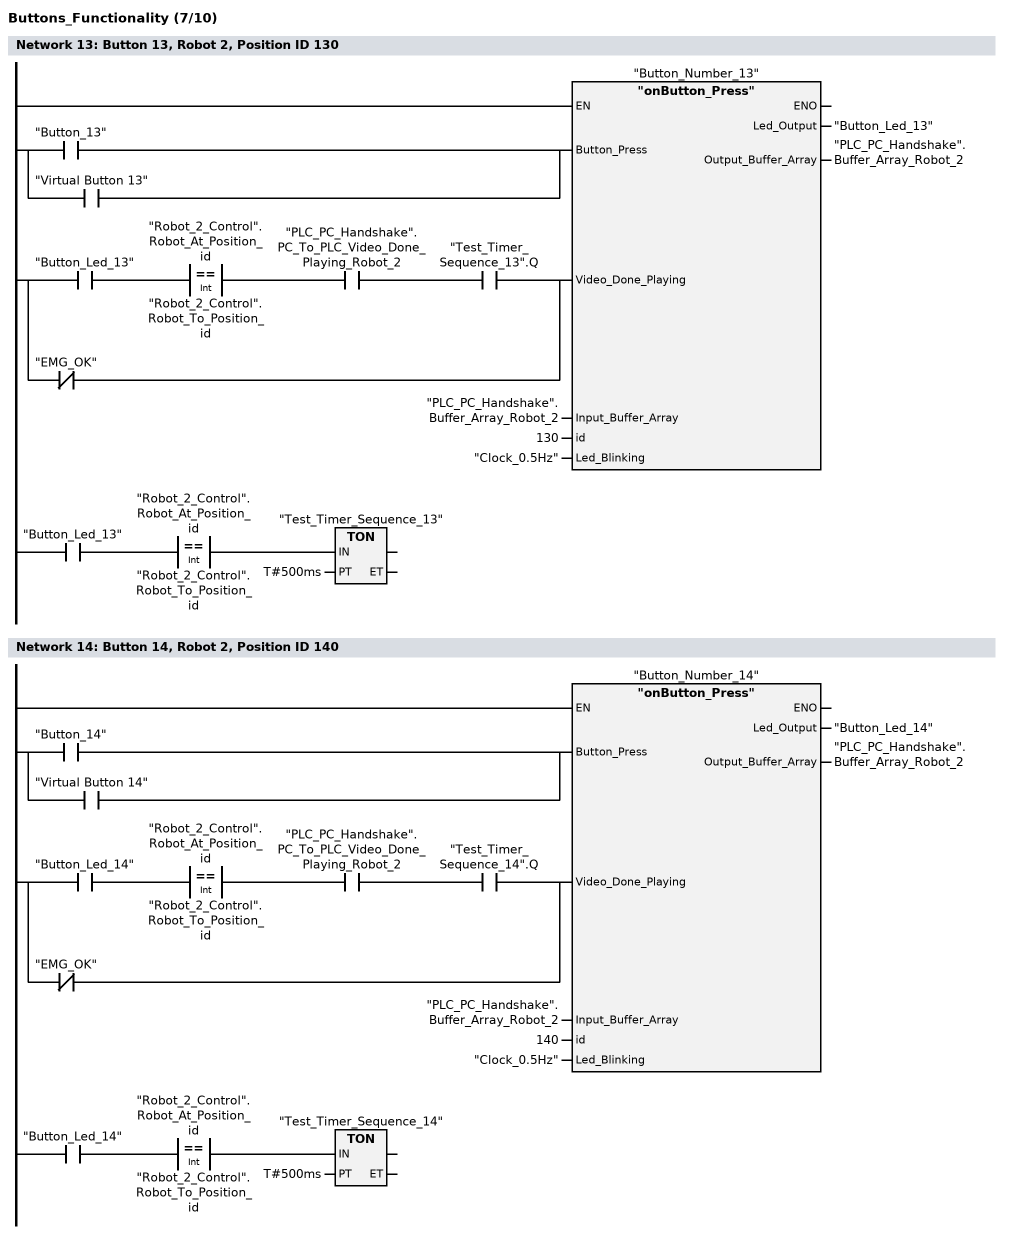
   "Button_Number_13"(Button_Press := "Button_13" OR "Virtual Button 13",   // "onButton_Press"
                      Video_Done_Playing := ("Button_Led_13" AND ("Robot_2_Control".Robot_At_Position_id = "Robot_2_Control".Robot_To_Position_id) AND "PLC_PC_Handshake".PC_To_PLC_Video_Done_Playing_Robot_2 AND "Test_Timer_Sequence_13".Q) OR NOT "EMG_OK",
                      Input_Buffer_Array := "PLC_PC_Handshake".Buffer_Array_Robot_2,
                      id := 130,
                      Led_Blinking := "Clock_0.5Hz",
                      Led_Output => "Button_Led_13",
                      Output_Buffer_Array => "PLC_PC_Handshake".Buffer_Array_Robot_2);
   "Test_Timer_Sequence_13".TON(IN := "Button_Led_13" AND ("Robot_2_Control".Robot_At_Position_id = "Robot_2_Control".Robot_To_Position_id),
                           PT := T#500ms);
END_REGION

REGION Network 14: Button 14, Robot 2, Position ID 140
   "Button_Number_14"(Button_Press := "Button_14" OR "Virtual Button 14",   // "onButton_Press"
                      Video_Done_Playing := ("Button_Led_14" AND ("Robot_2_Control".Robot_At_Position_id = "Robot_2_Control".Robot_To_Position_id) AND "PLC_PC_Handshake".PC_To_PLC_Video_Done_Playing_Robot_2 AND "Test_Timer_Sequence_14".Q) OR NOT "EMG_OK",
                      Input_Buffer_Array := "PLC_PC_Handshake".Buffer_Array_Robot_2,
                      id := 140,
                      Led_Blinking := "Clock_0.5Hz",
                      Led_Output => "Button_Led_14",
                      Output_Buffer_Array => "PLC_PC_Handshake".Buffer_Array_Robot_2);
   "Test_Timer_Sequence_14".TON(IN := "Button_Led_14" AND ("Robot_2_Control".Robot_At_Position_id = "Robot_2_Control".Robot_To_Position_id),
                           PT := T#500ms);
END_REGION

REGION Network 15: Button 15, Robot 2, Position ID 150
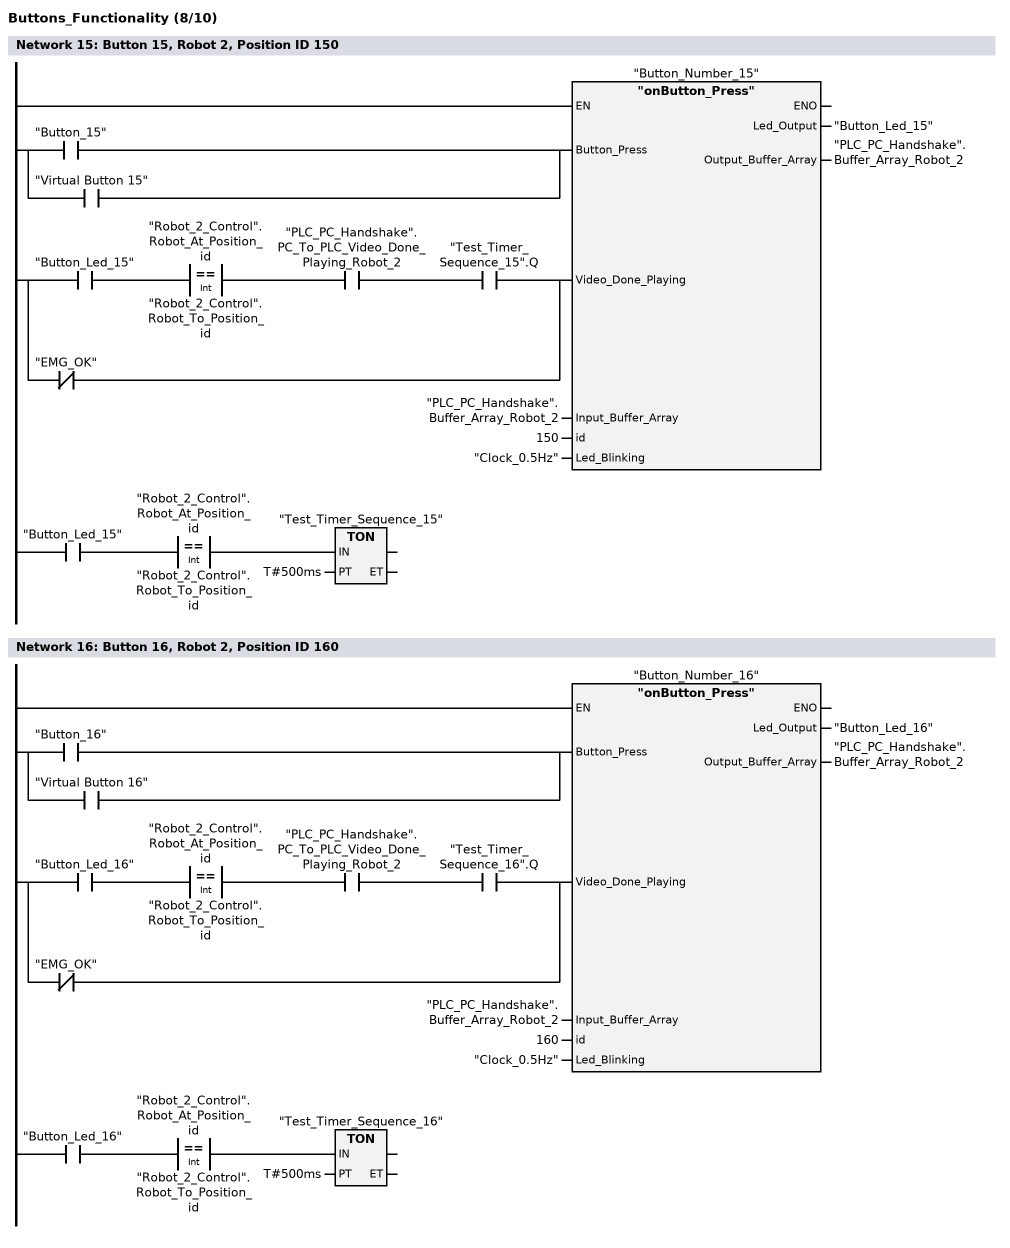
   "Button_Number_15"(Button_Press := "Button_15" OR "Virtual Button 15",   // "onButton_Press"
                      Video_Done_Playing := ("Button_Led_15" AND ("Robot_2_Control".Robot_At_Position_id = "Robot_2_Control".Robot_To_Position_id) AND "PLC_PC_Handshake".PC_To_PLC_Video_Done_Playing_Robot_2 AND "Test_Timer_Sequence_15".Q) OR NOT "EMG_OK",
                      Input_Buffer_Array := "PLC_PC_Handshake".Buffer_Array_Robot_2,
                      id := 150,
                      Led_Blinking := "Clock_0.5Hz",
                      Led_Output => "Button_Led_15",
                      Output_Buffer_Array => "PLC_PC_Handshake".Buffer_Array_Robot_2);
   "Test_Timer_Sequence_15".TON(IN := "Button_Led_15" AND ("Robot_2_Control".Robot_At_Position_id = "Robot_2_Control".Robot_To_Position_id),
                           PT := T#500ms);
END_REGION

REGION Network 16: Button 16, Robot 2, Position ID 160
   "Button_Number_16"(Button_Press := "Button_16" OR "Virtual Button 16",   // "onButton_Press"
                      Video_Done_Playing := ("Button_Led_16" AND ("Robot_2_Control".Robot_At_Position_id = "Robot_2_Control".Robot_To_Position_id) AND "PLC_PC_Handshake".PC_To_PLC_Video_Done_Playing_Robot_2 AND "Test_Timer_Sequence_16".Q) OR NOT "EMG_OK",
                      Input_Buffer_Array := "PLC_PC_Handshake".Buffer_Array_Robot_2,
                      id := 160,
                      Led_Blinking := "Clock_0.5Hz",
                      Led_Output => "Button_Led_16",
                      Output_Buffer_Array => "PLC_PC_Handshake".Buffer_Array_Robot_2);
   "Test_Timer_Sequence_16".TON(IN := "Button_Led_16" AND ("Robot_2_Control".Robot_At_Position_id = "Robot_2_Control".Robot_To_Position_id),
                           PT := T#500ms);
END_REGION

REGION Network 17: Button 17, Robot 2, Position ID 170
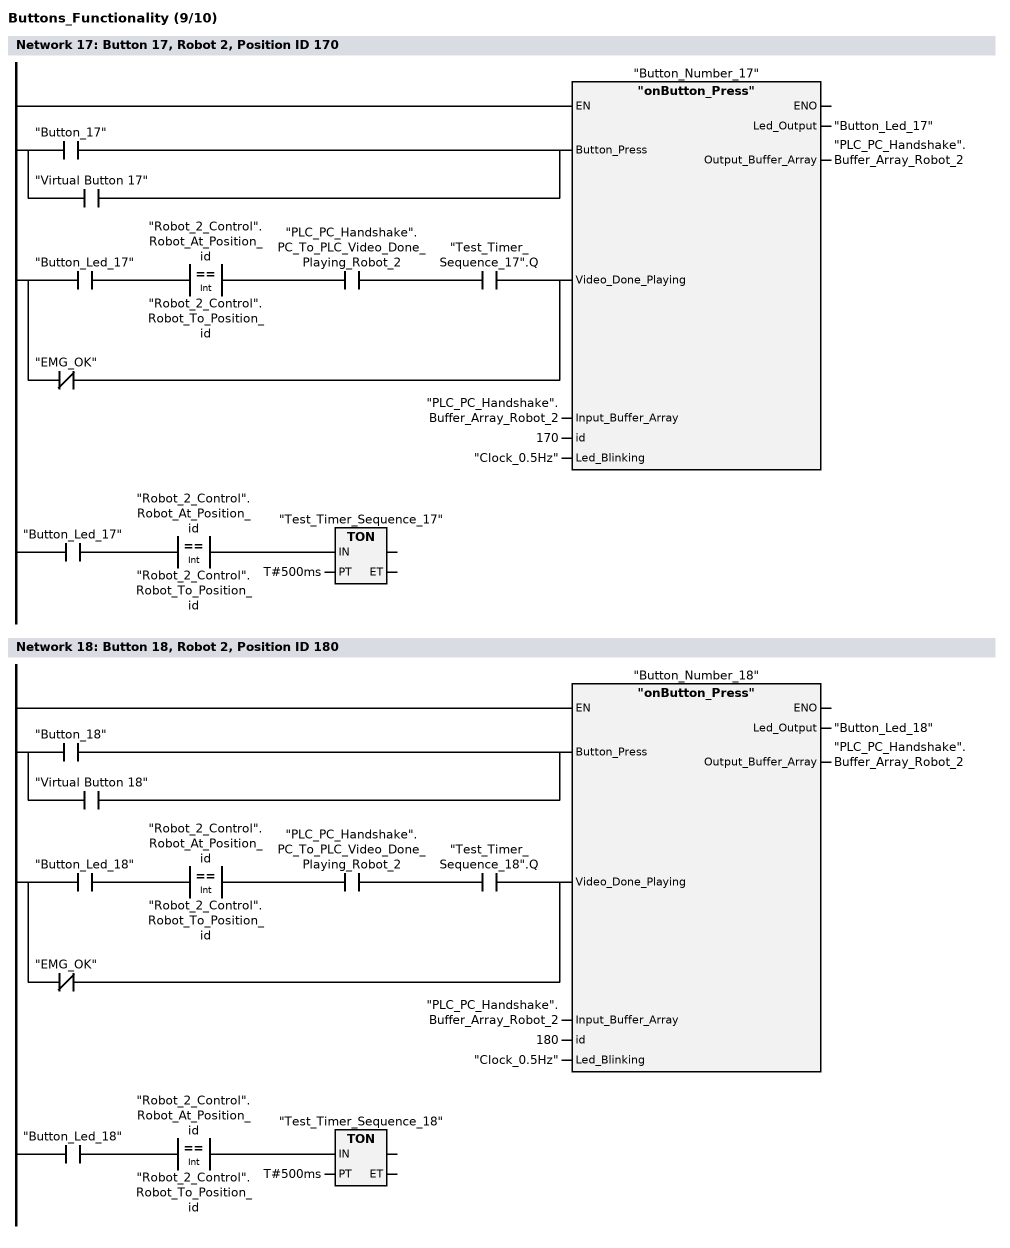
   "Button_Number_17"(Button_Press := "Button_17" OR "Virtual Button 17",   // "onButton_Press"
                      Video_Done_Playing := ("Button_Led_17" AND ("Robot_2_Control".Robot_At_Position_id = "Robot_2_Control".Robot_To_Position_id) AND "PLC_PC_Handshake".PC_To_PLC_Video_Done_Playing_Robot_2 AND "Test_Timer_Sequence_17".Q) OR NOT "EMG_OK",
                      Input_Buffer_Array := "PLC_PC_Handshake".Buffer_Array_Robot_2,
                      id := 170,
                      Led_Blinking := "Clock_0.5Hz",
                      Led_Output => "Button_Led_17",
                      Output_Buffer_Array => "PLC_PC_Handshake".Buffer_Array_Robot_2);
   "Test_Timer_Sequence_17".TON(IN := "Button_Led_17" AND ("Robot_2_Control".Robot_At_Position_id = "Robot_2_Control".Robot_To_Position_id),
                           PT := T#500ms);
END_REGION

REGION Network 18: Button 18, Robot 2, Position ID 180
   "Button_Number_18"(Button_Press := "Button_18" OR "Virtual Button 18",   // "onButton_Press"
                      Video_Done_Playing := ("Button_Led_18" AND ("Robot_2_Control".Robot_At_Position_id = "Robot_2_Control".Robot_To_Position_id) AND "PLC_PC_Handshake".PC_To_PLC_Video_Done_Playing_Robot_2 AND "Test_Timer_Sequence_18".Q) OR NOT "EMG_OK",
                      Input_Buffer_Array := "PLC_PC_Handshake".Buffer_Array_Robot_2,
                      id := 180,
                      Led_Blinking := "Clock_0.5Hz",
                      Led_Output => "Button_Led_18",
                      Output_Buffer_Array => "PLC_PC_Handshake".Buffer_Array_Robot_2);
   "Test_Timer_Sequence_18".TON(IN := "Button_Led_18" AND ("Robot_2_Control".Robot_At_Position_id = "Robot_2_Control".Robot_To_Position_id),
                           PT := T#500ms);
END_REGION

REGION Network 19: Reset Buffer Arrays
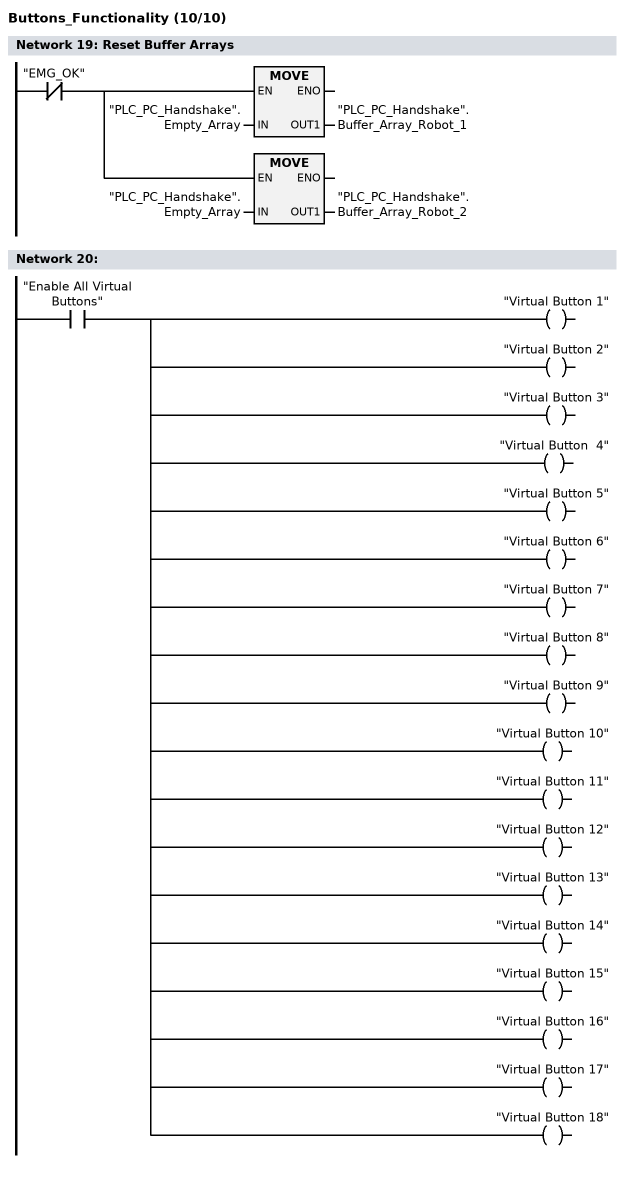
   RUNG wire#powerrail
      I_Contact( "EMG_OK" )
      wire#w1
      Move(in := "PLC_PC_Handshake".Empty_Array, out1 => "PLC_PC_Handshake".Buffer_Array_Robot_1)
   END_RUNG
   RUNG wire#w1
      Move(in := "PLC_PC_Handshake".Empty_Array, out1 => "PLC_PC_Handshake".Buffer_Array_Robot_2)
   END_RUNG
   // the same network as SCL:
   IF NOT "EMG_OK" THEN
       "PLC_PC_Handshake".Buffer_Array_Robot_1 := "PLC_PC_Handshake".Empty_Array;
       "PLC_PC_Handshake".Buffer_Array_Robot_2 := "PLC_PC_Handshake".Empty_Array;
   END_IF;
END_REGION

REGION Network 20
   RUNG wire#powerrail
      Contact( "Enable All Virtual Buttons" )
      wire#w1
      Coil( "Virtual Button 1" )
   END_RUNG
   RUNG wire#w1
      Coil( "Virtual Button 2" )
   END_RUNG
   RUNG wire#w1
      Coil( "Virtual Button 3" )
   END_RUNG
   RUNG wire#w1
      Coil( "Virtual Button  4" )
   END_RUNG
   RUNG wire#w1
      Coil( "Virtual Button 5" )
   END_RUNG
   RUNG wire#w1
      Coil( "Virtual Button 6" )
   END_RUNG
   RUNG wire#w1
      Coil( "Virtual Button 7" )
   END_RUNG
   RUNG wire#w1
      Coil( "Virtual Button 8" )
   END_RUNG
   RUNG wire#w1
      Coil( "Virtual Button 9" )
   END_RUNG
   RUNG wire#w1
      Coil( "Virtual Button 10" )
   END_RUNG
   RUNG wire#w1
      Coil( "Virtual Button 11" )
   END_RUNG
   RUNG wire#w1
      Coil( "Virtual Button 12" )
   END_RUNG
   RUNG wire#w1
      Coil( "Virtual Button 13" )
   END_RUNG
   RUNG wire#w1
      Coil( "Virtual Button 14" )
   END_RUNG
   RUNG wire#w1
      Coil( "Virtual Button 15" )
   END_RUNG
   RUNG wire#w1
      Coil( "Virtual Button 16" )
   END_RUNG
   RUNG wire#w1
      Coil( "Virtual Button 17" )
   END_RUNG
   RUNG wire#w1
      Coil( "Virtual Button 18" )
   END_RUNG
   // the same network as SCL:
   "Virtual Button 1" := "Enable All Virtual Buttons";
   "Virtual Button 2" := "Enable All Virtual Buttons";
   "Virtual Button 3" := "Enable All Virtual Buttons";
   "Virtual Button  4" := "Enable All Virtual Buttons";
   "Virtual Button 5" := "Enable All Virtual Buttons";
   "Virtual Button 6" := "Enable All Virtual Buttons";
   "Virtual Button 7" := "Enable All Virtual Buttons";
   "Virtual Button 8" := "Enable All Virtual Buttons";
   "Virtual Button 9" := "Enable All Virtual Buttons";
   "Virtual Button 10" := "Enable All Virtual Buttons";
   "Virtual Button 11" := "Enable All Virtual Buttons";
   "Virtual Button 12" := "Enable All Virtual Buttons";
   "Virtual Button 13" := "Enable All Virtual Buttons";
   "Virtual Button 14" := "Enable All Virtual Buttons";
   "Virtual Button 15" := "Enable All Virtual Buttons";
   "Virtual Button 16" := "Enable All Virtual Buttons";
   "Virtual Button 17" := "Enable All Virtual Buttons";
   "Virtual Button 18" := "Enable All Virtual Buttons";
END_REGION
END_FUNCTION

FUNCTION "Robots_Functionality" : Void   // FC3, LAD
{ S7_Optimized_Access := 'TRUE' }
VERSION : 0.1
BEGIN

REGION Network 1: Robot 1
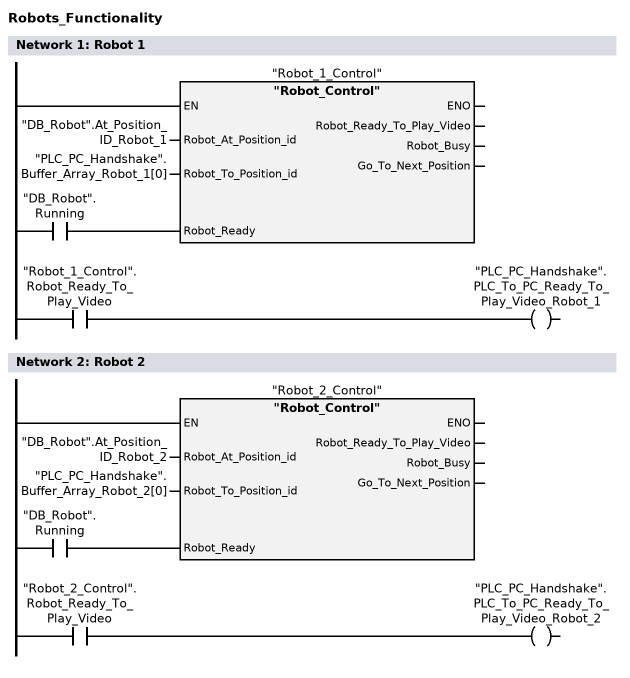
   RUNG wire#powerrail
      "Robot_1_Control"(Robot_Ready := wire#w1, Robot_At_Position_id := "DB_Robot".At_Position_ID_Robot_1, Robot_To_Position_id := "PLC_PC_Handshake".Buffer_Array_Robot_1[0], Robot_Ready_To_Play_Video =>, Robot_Busy =>, Go_To_Next_Position =>)
   END_RUNG
   RUNG wire#powerrail
      Contact( "DB_Robot".Running )
   END_RUNG wire#w1
   RUNG wire#powerrail
      Contact( "Robot_1_Control".Robot_Ready_To_Play_Video )
      Coil( "PLC_PC_Handshake".PLC_To_PC_Ready_To_Play_Video_Robot_1 )
   END_RUNG
   // the same network as SCL:
   "Robot_1_Control"(Robot_At_Position_id := "DB_Robot".At_Position_ID_Robot_1,   // "Robot_Control"
                     Robot_To_Position_id := "PLC_PC_Handshake".Buffer_Array_Robot_1[0],
                     Robot_Ready := "DB_Robot".Running);
   "PLC_PC_Handshake".PLC_To_PC_Ready_To_Play_Video_Robot_1 := "Robot_1_Control".Robot_Ready_To_Play_Video;
END_REGION

REGION Network 2: Robot 2
   RUNG wire#powerrail
      "Robot_2_Control"(Robot_Ready := wire#w1, Robot_At_Position_id := "DB_Robot".At_Position_ID_Robot_2, Robot_To_Position_id := "PLC_PC_Handshake".Buffer_Array_Robot_2[0], Robot_Ready_To_Play_Video =>, Robot_Busy =>, Go_To_Next_Position =>)
   END_RUNG
   RUNG wire#powerrail
      Contact( "DB_Robot".Running )
   END_RUNG wire#w1
   RUNG wire#powerrail
      Contact( "Robot_2_Control".Robot_Ready_To_Play_Video )
      Coil( "PLC_PC_Handshake".PLC_To_PC_Ready_To_Play_Video_Robot_2 )
   END_RUNG
   // the same network as SCL:
   "Robot_2_Control"(Robot_At_Position_id := "DB_Robot".At_Position_ID_Robot_2,   // "Robot_Control"
                     Robot_To_Position_id := "PLC_PC_Handshake".Buffer_Array_Robot_2[0],
                     Robot_Ready := "DB_Robot".Running);
   "PLC_PC_Handshake".PLC_To_PC_Ready_To_Play_Video_Robot_2 := "Robot_2_Control".Robot_Ready_To_Play_Video;
END_REGION
END_FUNCTION

FUNCTION "Robot Enable - Reset" : Void   // FC4, LAD
{ S7_Optimized_Access := 'TRUE' }
VERSION : 0.1
BEGIN

REGION Network 1: Input Data From Robot
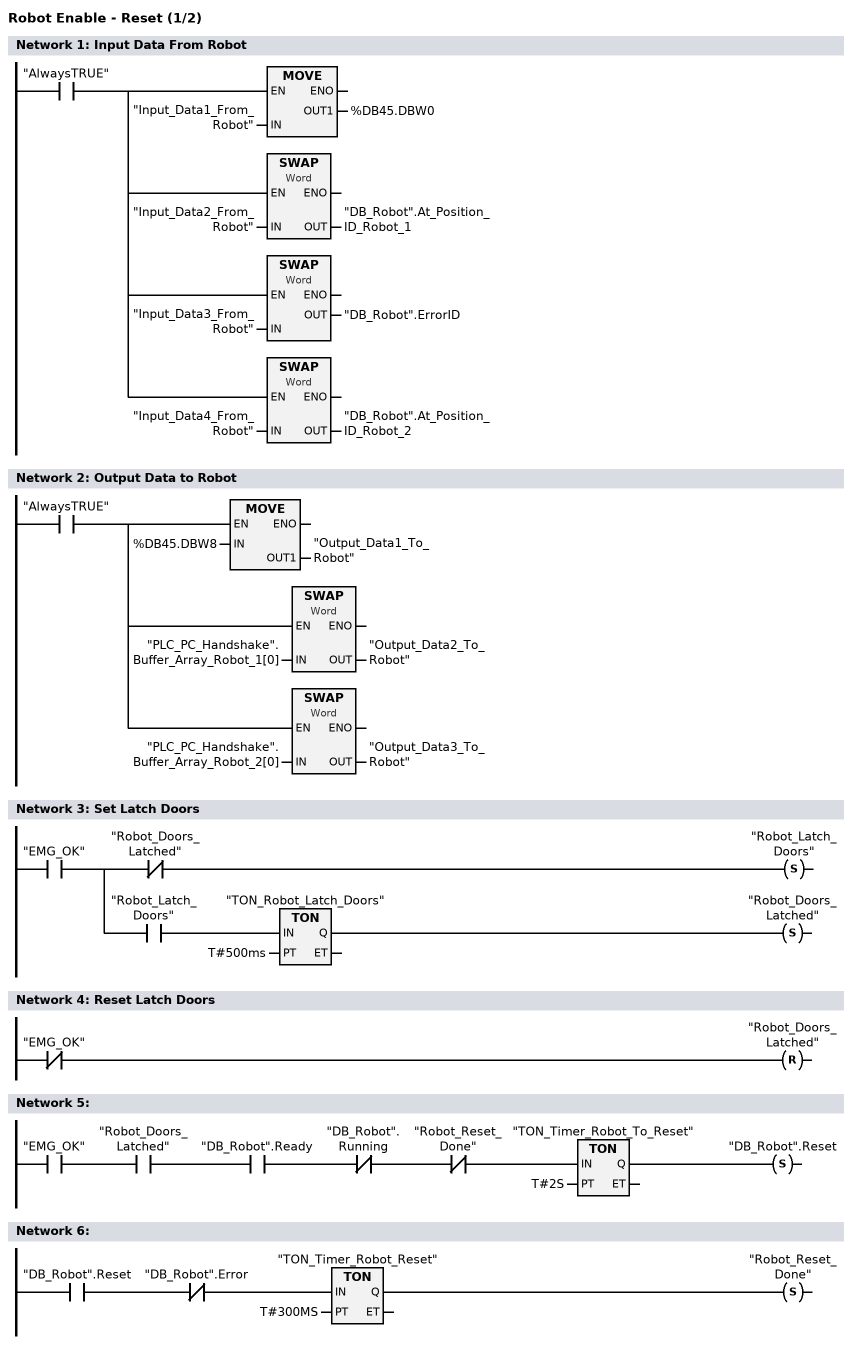
   IF "AlwaysTRUE" THEN
       %DB45.DBW0 := "Input_Data1_From_Robot";
       "DB_Robot".At_Position_ID_Robot_1 := SWAP("Input_Data2_From_Robot");
       "DB_Robot".ErrorID := SWAP("Input_Data3_From_Robot");
       "DB_Robot".At_Position_ID_Robot_2 := SWAP("Input_Data4_From_Robot");
   END_IF;
END_REGION

REGION Network 2: Output Data to Robot
   IF "AlwaysTRUE" THEN
       "Output_Data1_To_Robot" := %DB45.DBW8;
       "Output_Data2_To_Robot" := SWAP("PLC_PC_Handshake".Buffer_Array_Robot_1[0]);
       "Output_Data3_To_Robot" := SWAP("PLC_PC_Handshake".Buffer_Array_Robot_2[0]);
   END_IF;
END_REGION

REGION Network 3: Set Latch Doors
   IF "EMG_OK" AND NOT "Robot_Doors_Latched" THEN "Robot_Latch_Doors" := TRUE; END_IF;
   "TON_Robot_Latch_Doors".TON(IN := "EMG_OK" AND "Robot_Latch_Doors", PT := T#500ms);
   IF "TON_Robot_Latch_Doors".Q THEN "Robot_Doors_Latched" := TRUE; END_IF;
END_REGION

REGION Network 4: Reset Latch Doors
   RUNG wire#powerrail
      I_Contact( "EMG_OK" )
      R_Coil( "Robot_Doors_Latched" )
   END_RUNG
   // the same network as SCL:
   IF NOT "EMG_OK" THEN "Robot_Doors_Latched" := FALSE; END_IF;
END_REGION

REGION Network 5
   "TON_Timer_Robot_To_Reset".TON(IN := "EMG_OK" AND "Robot_Doors_Latched" AND "DB_Robot".Ready AND NOT "DB_Robot".Running AND NOT "Robot_Reset_Done",
                           PT := T#2S);
   IF "TON_Timer_Robot_To_Reset".Q THEN "DB_Robot".Reset := TRUE; END_IF;
END_REGION

REGION Network 6
   "TON_Timer_Robot_Reset".TON(IN := "DB_Robot".Reset AND NOT "DB_Robot".Error, PT := T#300MS);
   IF "TON_Timer_Robot_Reset".Q THEN "Robot_Reset_Done" := TRUE; END_IF;
END_REGION

REGION Network 7
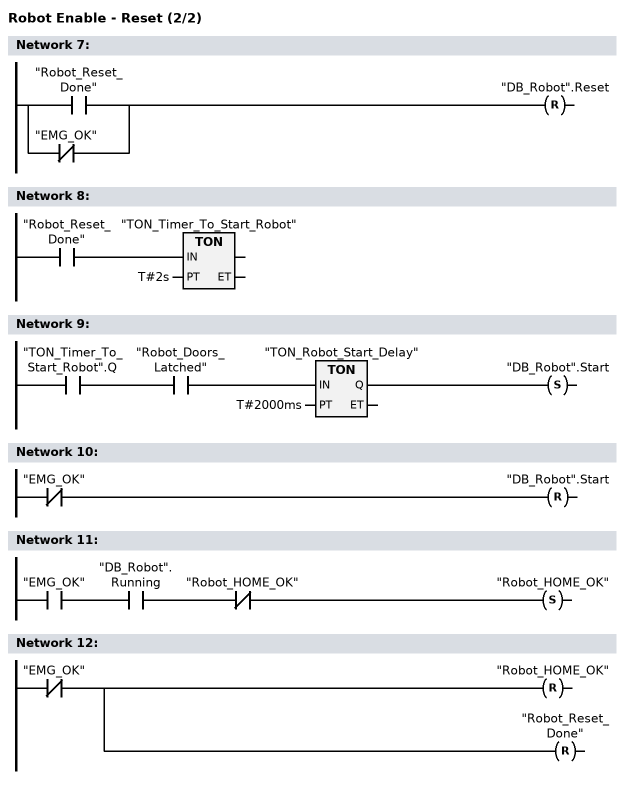
   RUNG wire#powerrail
      Contact( "Robot_Reset_Done" )
      wire#w1
      R_Coil( "DB_Robot".Reset )
   END_RUNG
   RUNG wire#powerrail
      I_Contact( "EMG_OK" )
   END_RUNG wire#w1
   // the same network as SCL:
   IF "Robot_Reset_Done" OR NOT "EMG_OK" THEN "DB_Robot".Reset := FALSE; END_IF;
END_REGION

REGION Network 8
   "TON_Timer_To_Start_Robot".TON(IN := "Robot_Reset_Done", PT := T#2s);
END_REGION

REGION Network 9
   "TON_Robot_Start_Delay".TON(IN := "TON_Timer_To_Start_Robot".Q AND "Robot_Doors_Latched", PT := T#2000ms);
   IF "TON_Robot_Start_Delay".Q THEN "DB_Robot".Start := TRUE; END_IF;
END_REGION

REGION Network 10
   RUNG wire#powerrail
      I_Contact( "EMG_OK" )
      R_Coil( "DB_Robot".Start )
   END_RUNG
   // the same network as SCL:
   IF NOT "EMG_OK" THEN "DB_Robot".Start := FALSE; END_IF;
END_REGION

REGION Network 11
   RUNG wire#powerrail
      Contact( "EMG_OK" )
      Contact( "DB_Robot".Running )
      I_Contact( "Robot_HOME_OK" )
      S_Coil( "Robot_HOME_OK" )
   END_RUNG
   // the same network as SCL:
   IF "EMG_OK" AND "DB_Robot".Running AND NOT "Robot_HOME_OK" THEN "Robot_HOME_OK" := TRUE; END_IF;
END_REGION

REGION Network 12
   RUNG wire#powerrail
      I_Contact( "EMG_OK" )
      wire#w1
      R_Coil( "Robot_HOME_OK" )
   END_RUNG
   RUNG wire#w1
      R_Coil( "Robot_Reset_Done" )
   END_RUNG
   // the same network as SCL:
   IF NOT "EMG_OK" THEN
       "Robot_HOME_OK" := FALSE;
       "Robot_Reset_Done" := FALSE;
   END_IF;
END_REGION
END_FUNCTION

ORGANIZATION_BLOCK "Main"   // OB1, LAD, ProgramCycle
TITLE = "Main Program Sweep (Cycle)"
{ S7_Optimized_Access := 'TRUE' }
VERSION : 0.1
   VAR_INPUT
      Initial_Call : Bool;   // Initial call of this OB
      Remanence : Bool;   // =True, if remanent data are available
   END_VAR
   VAR_TEMP
      tempIndex : Int;
   END_VAR
BEGIN

REGION Network 1: Manage PC To PLC Connection
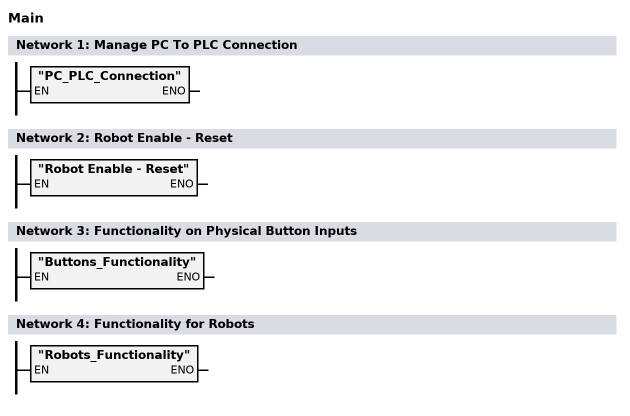
   RUNG wire#powerrail
      "PC_PLC_Connection"()
   END_RUNG
   // the same network as SCL:
   "PC_PLC_Connection"();
END_REGION

REGION Network 2: Robot Enable - Reset
   RUNG wire#powerrail
      "Robot Enable - Reset"()
   END_RUNG
   // the same network as SCL:
   "Robot Enable - Reset"();
END_REGION

REGION Network 3: Functionality on Physical Button Inputs
   RUNG wire#powerrail
      "Buttons_Functionality"()
   END_RUNG
   // the same network as SCL:
   "Buttons_Functionality"();
END_REGION

REGION Network 4: Functionality for Robots
   RUNG wire#powerrail
      "Robots_Functionality"()
   END_RUNG
   // the same network as SCL:
   "Robots_Functionality"();
END_REGION
END_ORGANIZATION_BLOCK

// folder: Functionalities

FUNCTION_BLOCK "onButton_Press"   // FB1, LAD
{ S7_Optimized_Access := 'TRUE' }
VERSION : 0.1
   VAR_INPUT
      Button_Press : Bool;
      Video_Done_Playing : Bool;
      Input_Buffer_Array : Array[0..19] of Int;
      id : Int;
      Led_Blinking : Bool;
   END_VAR
   VAR_OUTPUT
      Led_Output : Bool;
      Output_Buffer_Array : Array[0..19] of Int;
   END_VAR
   VAR
      Bit_State : Bool;
      temp_Buffer_Array : Array[0..19] of Int;
      Button_Trigger : Bool;
      Edit_Buffer : Bool;
      Video_Done_Trigger : Bool;
      Position_of_id_onBuffer : Int;
      Led_Flashes_Cnt : Int;
      Video_Done_Falling_Trigger_Pulse : F_TRIG;
      TOF_Enable_Led_Output : TOF_TIME;
      TON_Enable_Button_Output : TON_TIME;
      Enable_Output_To_Indicate_Priority : Bool;
      TON_Disable_Button_Output : TON_TIME;
      ResetTimers : Bool;
      Delay_Reset_Timers : TON_TIME;
      TEST_COUNTER : Int;
      TEST_BIT_COUNTER : Int;
   END_VAR
   VAR RETAIN
      Bit_Set_Counter : CTU_INT;
   END_VAR
   VAR_TEMP
      i : Int;
   END_VAR
   VAR_TEMP   // added for the SCL form of the ladder/FBD networks
      _w1 : Bool;
   END_VAR
BEGIN

REGION Network 1 (SCL): Assign Output Array equal to Input (Pass by value)
   #temp_Buffer_Array := #Input_Buffer_Array;
END_REGION

REGION Network 2: On Button Press set BitState to TRUE
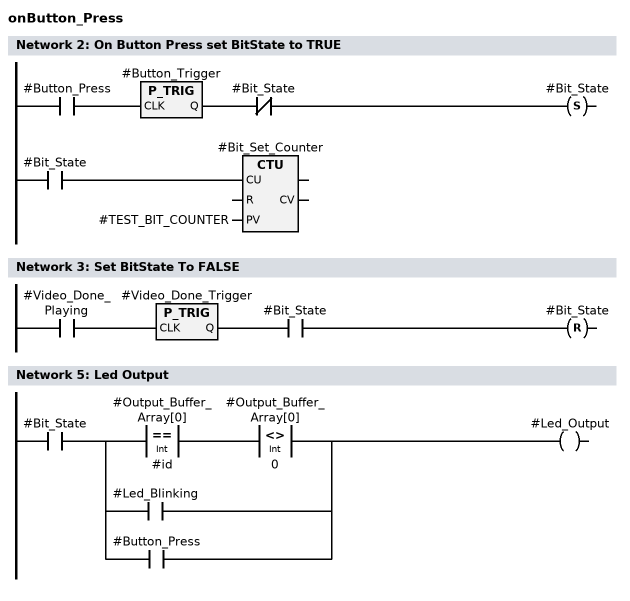
   #_w1 := #Button_Press AND NOT #Button_Trigger;   // rising edge
   #Button_Trigger := #Button_Press;
   IF #_w1 AND NOT #Bit_State THEN #Bit_State := TRUE; END_IF;
   #Bit_Set_Counter(CU := #Bit_State, PV := #TEST_BIT_COUNTER);   // CTU
END_REGION

REGION Network 3: Set BitState To FALSE
   RUNG wire#powerrail
      Contact( #Video_Done_Playing )
      P_Trig( #Video_Done_Trigger )
      Contact( #Bit_State )
      R_Coil( #Bit_State )
   END_RUNG
   // the same network as SCL:
   #_w1 := #Video_Done_Playing AND NOT #Video_Done_Trigger;   // rising edge
   #Video_Done_Trigger := #Video_Done_Playing;
   IF #_w1 AND #Bit_State THEN #Bit_State := FALSE; END_IF;
END_REGION

REGION Network 4 (SCL): Buffer Array

   IF (#Bit_State) THEN //IF BUTTON IS PRESSED



       #Edit_Buffer := FALSE;

       IF (#temp_Buffer_Array[0] = #id) THEN // CHECK IF THE FIRST ELEMENT OF THE ARRAY HOLDS THE CURRENT #id NUMBER
           #Position_of_id_onBuffer := 0;
       ELSE
           FOR #i := 0 TO 19 DO //CHECK BUFFER ARRAY 
               IF (#temp_Buffer_Array[#i] = #id) THEN //FIND THE POSITION OF THE #id ON THE ARRAY        
                   #Position_of_id_onBuffer := #i;
                   EXIT; 
               ELSIF (#temp_Buffer_Array[#i] = 0) THEN // ELSE PLACE THE ID ON THE FIRST FREE SLOT OF THE ARRAY (=0)
                   #temp_Buffer_Array[#i] := #id;
                   EXIT; 
               END_IF;
           END_FOR;
       END_IF; //END OF CHECK BUFFER ARRAY

   ELSIF (#Bit_State = FALSE AND #Edit_Buffer = FALSE) THEN //WHEN PLAYING THE VIDEO IS DONE, RESET BIT STATE AND REMOVE ELEMENT FROM BUFFER

       #Edit_Buffer := TRUE;

       #TEST_COUNTER := 0;
       FOR #i := 0 TO 19 DO  //SHIFT LEFT ALL ELEMENETS OF THE ARRAY EXCEPT OF THE LAST ONE WHICH IS EQUAL TO 0 (PREVENT ARRAY OUT OF INDEX ERROR)
           IF (#i <> 19) THEN
               #temp_Buffer_Array[#i] := #temp_Buffer_Array[#i + 1];
           ELSE
               #temp_Buffer_Array[#i] := 0;
           END_IF;

           #TEST_COUNTER := #TEST_COUNTER + 1;
       END_FOR;

   END_IF;
END_REGION

REGION Network 5: Led Output
   RUNG wire#powerrail
      Contact( #Bit_State )
      wire#w1
      { S7_Templates := "SrcType := Int" } EQ_Contact(in1 := #Output_Buffer_Array[0], in2 := #id)
      { S7_Templates := "SrcType := Int" } NE_Contact(in1 := #Output_Buffer_Array[0], in2 := 0)
      wire#w2
      Coil( #Led_Output )
   END_RUNG
   RUNG wire#w1
      Contact( #Led_Blinking )
   END_RUNG wire#w2
   RUNG wire#w1
      Contact( #Button_Press )
   END_RUNG wire#w2
   // the same network as SCL:
   #Led_Output := #Bit_State AND (((#Output_Buffer_Array[0] = #id) AND (#Output_Buffer_Array[0] <> 0)) OR #Led_Blinking OR #Button_Press);
END_REGION

REGION Network 6 (SCL)
   #Output_Buffer_Array := #temp_Buffer_Array;
END_REGION
END_FUNCTION_BLOCK

FUNCTION_BLOCK "Robot_Control"   // FB2, SCL
{ S7_Optimized_Access := 'TRUE' }
VERSION : 0.1
   VAR_INPUT
      Robot_At_Position_id : Int;
      Robot_To_Position_id : Int;
      Robot_Ready : Bool;
   END_VAR
   VAR_OUTPUT
      Robot_Ready_To_Play_Video : Bool;
      Robot_Busy : Bool;
      Go_To_Next_Position : Bool;
   END_VAR
BEGIN
   IF #Robot_At_Position_id <> #Robot_To_Position_id AND #Robot_To_Position_id <> 0 THEN //GO TO POSITION OF THE ID
       #Robot_Busy := TRUE;
       #Go_To_Next_Position := TRUE;
       #Robot_Ready_To_Play_Video := FALSE;
   END_IF;

   IF #Robot_At_Position_id = #Robot_To_Position_id AND #Robot_Busy = TRUE AND #Robot_At_Position_id <> 0 THEN //READY TO PLAY VIDEO
       #Go_To_Next_Position := FALSE;
       #Robot_Ready_To_Play_Video := TRUE;
   END_IF;

   IF #Robot_At_Position_id = 0 THEN
       #Robot_Ready_To_Play_Video := FALSE;
   END_IF;

   IF #Robot_At_Position_id = #Robot_To_Position_id AND #Robot_To_Position_id = 0 THEN //NO NEW BUTTON IS PRESSED, BUFFER ARRAY IS EMPTY
       #Robot_Busy := FALSE;
   END_IF;
END_FUNCTION_BLOCK